# B&R Automation Studio project MotionTestBenchMaster (part 45)

#### HmiInterfacesNew.st
```iecst
ACTION HmiInterfacesNew:
	xAxisInVelocityControl	:= FALSE;

	IF VAR_Machine.iq_stParameter.i_uiAxisSelected >= CST_FillerSubModuleHmiStart AND VAR_Machine.iq_stParameter.i_uiAxisSelected <= CST_FillerSubModuleHmiStart + CST_LastFillerModuleAxis	THEN
		VAR_Machine.stFillerModule.iq_stParameters.i_uiAxisSelected	:= VAR_Machine.iq_stParameter.i_uiAxisSelected - CST_FillerSubModuleHmiStart;
	ELSIF VAR_Machine.iq_stParameter.i_uiAxisSelected >= CST_OutletSubModuleHmiStart AND VAR_Machine.iq_stParameter.i_uiAxisSelected <= CST_OutletSubModuleHmiStart + CST_LastOutletModuleAxis THEN
		VAR_Machine.stOutletModule.iq_stParameters.i_uiAxisSelected	:= VAR_Machine.iq_stParameter.i_uiAxisSelected - CST_OutletSubModuleHmiStart;
	ELSIF VAR_Machine.iq_stParameter.i_uiAxisSelected >= CST_InletSubModuleHmiStart AND VAR_Machine.iq_stParameter.i_uiAxisSelected <= CST_InletSubModuleHmiStart + CST_LastInletModuleAxis THEN
		VAR_Machine.stInletModule.iq_stParameters.i_uiAxisSelected	:= VAR_Machine.iq_stParameter.i_uiAxisSelected - CST_InletSubModuleHmiStart;
	ELSIF VAR_Machine.iq_stParameter.i_uiAxisSelected = CST_MachinePhasingOffset THEN
		VAR_Machine.stMasterModule.iq_stParameters.i_uiAxisSelected	:=	VAR_Machine.iq_stParameter.i_uiAxisSelected;
	END_IF
	////////////////////////////////////////////////

	HMI_MC_GenericAxisDataNew[1].uiDiagCode				:= VAR_Machine.stMasterModule.iq_astSubModuleAxis[CST_MachineMasterAxis].iq_stStatus.q_stMainAxisStatus.q_stInfo.Diag.StatusID.Code;
	HMI_MC_GenericAxisDataNew[1].rLagError				:= FC_DegreeToMm(CFG_MC.Mechanical.MachineStep, VAR_Machine.stMasterModule.iq_astSubModuleAxis[CST_MachineMasterAxis].iq_stStatus.q_stMainAxisStatus.q_rLagError,FALSE);

	HMI_MC_GenericAxisDataNew[1].xMotorWithBrake		:= VAR_Machine.stMasterModule.iq_astSubModuleAxis[CST_MachineMasterAxis].iq_stStatus.q_stMainAxisStatus.q_xMotorWithBrake;
	HMI_MC_GenericAxisDataNew[1].xThirdPartMotor		:= VAR_Machine.stMasterModule.iq_astSubModuleAxis[CST_MachineMasterAxis].iq_stStatus.q_stMainAxisStatus.q_xThirdPartyMotor;
	HMI_MC_GenericAxisDataNew[1].xVelocityControl		:= VAR_Machine.stMasterModule.iq_astSubModuleAxis[CST_MachineMasterAxis].iq_stStatus.q_stMainAxisStatus.q_xVelocityControl;
	HMI_MC_GenericAxisDataNew[1].xInduction				:= VAR_Machine.stMasterModule.iq_astSubModuleAxis[CST_MachineMasterAxis].iq_stStatus.q_stMainAxisStatus.q_xInduction;
	HMI_MC_GenericAxisDataNew[1].rHomingOffset			:= VAR_Machine.stMasterModule.iq_astSubModuleAxis[CST_MachineMasterAxis].iq_stStatus.q_stMainAxisStatus.q_rHomingOffset;

	HMI_MC_GenericAxisDataNew[1].rPosition				:= LREAL_TO_REAL(VAR_Machine.stMasterModule.iq_astSubModuleAxis[CST_MachineMasterAxis].iq_stStatus.q_stMainAxisStatus.q_lrPosition);
	HMI_MC_GenericAxisDataNew[1].rPosition_mm			:= FC_DegreeToMm(CFG_MC.Mechanical.MachineStep,HMI_MC_GenericAxisDataNew[1].rPosition,TRUE);//V1.7.2

	HMI_MC_GenericAxisDataNew[1].rVelocity				:= VAR_Machine.stMasterModule.iq_astSubModuleAxis[CST_MachineMasterAxis].iq_stStatus.q_stMainAxisStatus.q_rVelocity * 10.0;

	HMI_MC_GenericAxisDataNew[1].rTotalPhasingOffset	:= FC_DegreeToMm(CFG_MC.Mechanical.MachineStep,VAR_Machine.stMasterModule.iq_astSubModuleAxis[CST_MachineMasterAxis].iq_stStatus.q_stMainAxisStatus.q_rTotalOffset,FALSE);

	HMI_MC_GenericAxisDataNew[1].xInitialized			:= VAR_Machine.stMasterModule.iq_astSubModuleAxis[CST_MachineMasterAxis].iq_stStatus.q_stMainAxisStatus.q_xInitDone;

	xPhasingRunning									:= VAR_Machine.stMasterModule.iq_astSubModuleAxis[CST_MachineMasterAxis].iq_stStatus.q_stMainAxisStatus.q_xPhasingRunning;

	IF HMI_MC_GenericAxisDataNew[1].xInitialized THEN
		HMI_MC_GenericAxisDataNew[1].xActive				:= VAR_Machine.stMasterModule.iq_astSubModuleAxis[CST_MachineMasterAxis].iq_stStatus.q_stMainAxisStatus.q_xActive;
		HMI_MC_GenericAxisDataNew[1].xBrakeReleased		:= FALSE;
		HMI_MC_GenericAxisDataNew[1].xEnabled;
		HMI_MC_GenericAxisDataNew[1].xFollowingError		:= FALSE;
		HMI_MC_GenericAxisDataNew[1].xHomed				:= FALSE;
		HMI_MC_GenericAxisDataNew[1].xInError				:= VAR_Machine.stMasterModule.iq_astSubModuleAxis[CST_MachineMasterAxis].iq_stStatus.q_stMainAxisStatus.q_xError;
		HMI_MC_GenericAxisDataNew[1].xInPosition			:= VAR_Machine.stMasterModule.iq_astSubModuleAxis[CST_MachineMasterAxis].iq_stStatus.q_stMainAxisStatus.q_xInPosition;
		HMI_MC_GenericAxisDataNew[1].xPowered				:= FALSE;
		HMI_MC_GenericAxisDataNew[1].xReal				:= FALSE;
		HMI_MC_GenericAxisDataNew[1].xRunning				:= FALSE;
		HMI_MC_GenericAxisDataNew[1].xSynchro				:= VAR_Machine.stMasterModule.iq_astSubModuleAxis[CST_MachineMasterAxis].iq_stStatus.q_stMainAxisStatus.q_xSynchronized;
		HMI_MC_GenericAxisDataNew[1].xTorqueError			:= FALSE;
		//			HMI_MC_GenericAxisDataNew[1].xHmiWait				:= FALSE;//V1.7.2
	ELSE
		HMI_MC_GenericAxisDataNew[1].xActive				:= FALSE;
		HMI_MC_GenericAxisDataNew[1].xBrakeReleased		:= FALSE;
		HMI_MC_GenericAxisDataNew[1].xEnabled;
		HMI_MC_GenericAxisDataNew[1].xFollowingError		:= FALSE;
		HMI_MC_GenericAxisDataNew[1].xHomed				:= FALSE;
		HMI_MC_GenericAxisDataNew[1].xInError				:= FALSE;
		HMI_MC_GenericAxisDataNew[1].xInPosition			:= FALSE;
		HMI_MC_GenericAxisDataNew[1].xPowered				:= FALSE;
		HMI_MC_GenericAxisDataNew[1].xReal				:= FALSE;
		HMI_MC_GenericAxisDataNew[1].xRunning				:= FALSE;
		HMI_MC_GenericAxisDataNew[1].xSynchro				:= FALSE;
		HMI_MC_GenericAxisDataNew[1].xTorqueError			:= FALSE;
		//			HMI_MC_GenericAxisDataNew[1].xHmiWait				:= TRUE;//v1.7.2
	END_IF

	FOR HMI_AxisIndex := 2 TO 14 DO //vrma
		//Inlet Axis Motor
		IF HMI_MC_GenericAxisDataNew[HMI_AxisIndex].uiAxisID >= CST_InletSubModuleHmiStart AND HMI_MC_GenericAxisDataNew[HMI_AxisIndex].uiAxisID <= CST_InletSubModuleHmiStart + CST_LastInletModuleAxis THEN

			HMI_MC_GenericAxisDataNew[HMI_AxisIndex].uiDiagCode				:= VAR_Machine.stInletModule.iq_astSubModuleAxis[HMI_MC_GenericAxisDataNew[HMI_AxisIndex].uiAxisID-CST_InletSubModuleHmiStart].iq_stStatus.q_stMainAxisStatus.q_stInfo.Diag.StatusID.Code;
			HMI_MC_GenericAxisDataNew[HMI_AxisIndex].iNextAx_Number;
			HMI_MC_GenericAxisDataNew[HMI_AxisIndex].iPrevAx_Number;
			HMI_MC_GenericAxisDataNew[HMI_AxisIndex].rEncoderTemperature		:= VAR_Machine.stInletModule.iq_astSubModuleAxis[HMI_MC_GenericAxisDataNew[HMI_AxisIndex].uiAxisID-CST_InletSubModuleHmiStart].iq_stStatus.q_stMainAxisStatus.q_rEncoderTemperature;
			HMI_MC_GenericAxisDataNew[HMI_AxisIndex].rMaxTorque;
			HMI_MC_GenericAxisDataNew[HMI_AxisIndex].rLagError				:= FC_DegreeToMm(CFG_MC.Mechanical.MachineStep, VAR_Machine.stInletModule.iq_astSubModuleAxis[HMI_MC_GenericAxisDataNew[HMI_AxisIndex].uiAxisID-CST_InletSubModuleHmiStart].iq_stStatus.q_stMainAxisStatus.q_rLagError, FALSE);

			HMI_MC_GenericAxisDataNew[HMI_AxisIndex].xMotorWithBrake			:= VAR_Machine.stInletModule.iq_astSubModuleAxis[HMI_MC_GenericAxisDataNew[HMI_AxisIndex].uiAxisID-CST_InletSubModuleHmiStart].iq_stStatus.q_stMainAxisStatus.q_xMotorWithBrake;
			HMI_MC_GenericAxisDataNew[HMI_AxisIndex].xThirdPartMotor			:= VAR_Machine.stInletModule.iq_astSubModuleAxis[HMI_MC_GenericAxisDataNew[HMI_AxisIndex].uiAxisID-CST_InletSubModuleHmiStart].iq_stStatus.q_stMainAxisStatus.q_xThirdPartyMotor;
			HMI_MC_GenericAxisDataNew[HMI_AxisIndex].xVelocityControl			:= VAR_Machine.stInletModule.iq_astSubModuleAxis[HMI_MC_GenericAxisDataNew[HMI_AxisIndex].uiAxisID-CST_InletSubModuleHmiStart].iq_stStatus.q_stMainAxisStatus.q_xVelocityControl;
			HMI_MC_GenericAxisDataNew[HMI_AxisIndex].xInduction				:= VAR_Machine.stInletModule.iq_astSubModuleAxis[HMI_MC_GenericAxisDataNew[HMI_AxisIndex].uiAxisID-CST_InletSubModuleHmiStart].iq_stStatus.q_stMainAxisStatus.q_xInduction;
			HMI_MC_GenericAxisDataNew[HMI_AxisIndex].rHomingOffset			:= VAR_Machine.stInletModule.iq_astSubModuleAxis[HMI_MC_GenericAxisDataNew[HMI_AxisIndex].uiAxisID-CST_InletSubModuleHmiStart].iq_stStatus.q_stMainAxisStatus.q_rHomingOffset;

			HMI_MC_GenericAxisDataNew[HMI_AxisIndex].rMotorTemperature		:= VAR_Machine.stInletModule.iq_astSubModuleAxis[HMI_MC_GenericAxisDataNew[HMI_AxisIndex].uiAxisID-CST_InletSubModuleHmiStart].iq_stStatus.q_stMainAxisStatus.q_rMotorTemperature;
			HMI_MC_GenericAxisDataNew[HMI_AxisIndex].rNextAx_Position_mm;
			HMI_MC_GenericAxisDataNew[HMI_AxisIndex].rPosition				:= LREAL_TO_REAL(VAR_Machine.stInletModule.iq_astSubModuleAxis[HMI_MC_GenericAxisDataNew[HMI_AxisIndex].uiAxisID-CST_InletSubModuleHmiStart].iq_stStatus.q_stMainAxisStatus.q_lrPosition);
			HMI_MC_GenericAxisDataNew[HMI_AxisIndex].rPosition_mm			:= FC_DegreeToMm(CFG_MC.Mechanical.MachineStep,HMI_MC_GenericAxisDataNew[HMI_AxisIndex].rPosition,TRUE);//v1.7.2

			HMI_MC_GenericAxisDataNew[HMI_AxisIndex].rPrevAx_Position_mm;
			HMI_MC_GenericAxisDataNew[HMI_AxisIndex].rTorque					:= LREAL_TO_REAL(VAR_Machine.stInletModule.iq_astSubModuleAxis[HMI_MC_GenericAxisDataNew[HMI_AxisIndex].uiAxisID-CST_InletSubModuleHmiStart].iq_stStatus.q_stMainAxisStatus.q_lrTorque);
			HMI_MC_GenericAxisDataNew[HMI_AxisIndex].rVelocity				:= VAR_Machine.stInletModule.iq_astSubModuleAxis[HMI_MC_GenericAxisDataNew[HMI_AxisIndex].uiAxisID-CST_InletSubModuleHmiStart].iq_stStatus.q_stMainAxisStatus.q_rVelocity * 10.0;
			HMI_MC_GenericAxisDataNew[HMI_AxisIndex].rSwitchValue;

			HMI_MC_GenericAxisDataNew[HMI_AxisIndex].rTotalPhasingOffset		:= FC_DegreeToMm(CFG_MC.Mechanical.MachineStep,VAR_Machine.stInletModule.iq_astSubModuleAxis[HMI_MC_GenericAxisDataNew[HMI_AxisIndex].uiAxisID-CST_InletSubModuleHmiStart].iq_stStatus.q_stMainAxisStatus.q_rTotalOffset,FALSE);

			HMI_MC_GenericAxisDataNew[HMI_AxisIndex].xInitialized				:= VAR_Machine.stInletModule.iq_astSubModuleAxis[HMI_MC_GenericAxisDataNew[HMI_AxisIndex].uiAxisID-CST_InletSubModuleHmiStart].iq_stStatus.q_stMainAxisStatus.q_xInitDone;

			xPhasingRunning									:= VAR_Machine.stInletModule.iq_astSubModuleAxis[HMI_MC_GenericAxisDataNew[HMI_AxisIndex].uiAxisID-CST_InletSubModuleHmiStart].iq_stStatus.q_stMainAxisStatus.q_xPhasingRunning;

			IF HMI_MC_GenericAxisDataNew[HMI_AxisIndex].xInitialized THEN
				HMI_MC_GenericAxisDataNew[HMI_AxisIndex].xActive				:= VAR_Machine.stInletModule.iq_astSubModuleAxis[HMI_MC_GenericAxisDataNew[HMI_AxisIndex].uiAxisID-CST_InletSubModuleHmiStart].iq_stStatus.q_stMainAxisStatus.q_xActive;
				HMI_MC_GenericAxisDataNew[HMI_AxisIndex].xBrakeReleased		:= VAR_Machine.stInletModule.iq_astSubModuleAxis[HMI_MC_GenericAxisDataNew[HMI_AxisIndex].uiAxisID-CST_InletSubModuleHmiStart].iq_stStatus.q_stMainAxisStatus.q_xBrakeReleased;
				HMI_MC_GenericAxisDataNew[HMI_AxisIndex].xEnabled;
				HMI_MC_GenericAxisDataNew[HMI_AxisIndex].xFollowingError		:= VAR_Machine.stInletModule.iq_astSubModuleAxis[HMI_MC_GenericAxisDataNew[HMI_AxisIndex].uiAxisID-CST_InletSubModuleHmiStart].iq_stStatus.q_stMainAxisStatus.q_xLagError;
				HMI_MC_GenericAxisDataNew[HMI_AxisIndex].xHomed				:= VAR_Machine.stInletModule.iq_astSubModuleAxis[HMI_MC_GenericAxisDataNew[HMI_AxisIndex].uiAxisID-CST_InletSubModuleHmiStart].iq_stStatus.q_stMainAxisStatus.q_xIsHomed;
				HMI_MC_GenericAxisDataNew[HMI_AxisIndex].xInError				:= VAR_Machine.stInletModule.iq_astSubModuleAxis[HMI_MC_GenericAxisDataNew[HMI_AxisIndex].uiAxisID-CST_InletSubModuleHmiStart].iq_stStatus.q_stMainAxisStatus.q_xError;
				HMI_MC_GenericAxisDataNew[HMI_AxisIndex].xInPosition			:= VAR_Machine.stInletModule.iq_astSubModuleAxis[HMI_MC_GenericAxisDataNew[HMI_AxisIndex].uiAxisID-CST_InletSubModuleHmiStart].iq_stStatus.q_stMainAxisStatus.q_xInPosition;
				HMI_MC_GenericAxisDataNew[HMI_AxisIndex].xPowered				:= VAR_Machine.stInletModule.iq_astSubModuleAxis[HMI_MC_GenericAxisDataNew[HMI_AxisIndex].uiAxisID-CST_InletSubModuleHmiStart].iq_stStatus.q_stMainAxisStatus.q_xPoweredOn;
				HMI_MC_GenericAxisDataNew[HMI_AxisIndex].xReal				:= VAR_Machine.stInletModule.iq_astSubModuleAxis[HMI_MC_GenericAxisDataNew[HMI_AxisIndex].uiAxisID-CST_InletSubModuleHmiStart].iq_stStatus.q_stMainAxisStatus.q_xAxisReal;
				HMI_MC_GenericAxisDataNew[HMI_AxisIndex].xRunning				:= NOT VAR_Machine.stInletModule.iq_astSubModuleAxis[HMI_MC_GenericAxisDataNew[HMI_AxisIndex].uiAxisID-CST_InletSubModuleHmiStart].iq_stStatus.q_stMainAxisStatus.q_xStopped;
				HMI_MC_GenericAxisDataNew[HMI_AxisIndex].xSynchro				:= VAR_Machine.stInletModule.iq_astSubModuleAxis[HMI_MC_GenericAxisDataNew[HMI_AxisIndex].uiAxisID-CST_InletSubModuleHmiStart].iq_stStatus.q_stMainAxisStatus.q_xSynchronized;
				HMI_MC_GenericAxisDataNew[HMI_AxisIndex].xTorqueError			:= VAR_Machine.stInletModule.iq_astSubModuleAxis[HMI_MC_GenericAxisDataNew[HMI_AxisIndex].uiAxisID-CST_InletSubModuleHmiStart].iq_stStatus.q_stMainAxisStatus.q_xTorqueError;
				//HMI_MC_GenericAxisDataNew[HMI_AxisIndex].xHmiWait				:= FALSE;//v1.7.2
			ELSE
				HMI_MC_GenericAxisDataNew[HMI_AxisIndex].xActive				:= FALSE;
				HMI_MC_GenericAxisDataNew[HMI_AxisIndex].xBrakeReleased		:= FALSE;
				HMI_MC_GenericAxisDataNew[HMI_AxisIndex].xEnabled;
				HMI_MC_GenericAxisDataNew[HMI_AxisIndex].xFollowingError		:= FALSE;
				HMI_MC_GenericAxisDataNew[HMI_AxisIndex].xHomed					:= FALSE;
				HMI_MC_GenericAxisDataNew[HMI_AxisIndex].xInError				:= FALSE;
				HMI_MC_GenericAxisDataNew[HMI_AxisIndex].xInPosition			:= FALSE;
				HMI_MC_GenericAxisDataNew[HMI_AxisIndex].xPowered				:= FALSE;
				HMI_MC_GenericAxisDataNew[HMI_AxisIndex].xReal					:= FALSE;
				HMI_MC_GenericAxisDataNew[HMI_AxisIndex].xRunning				:= FALSE;
				HMI_MC_GenericAxisDataNew[HMI_AxisIndex].xSynchro				:= FALSE;
				HMI_MC_GenericAxisDataNew[HMI_AxisIndex].xTorqueError			:= FALSE;
				//				HMI_MC_GenericAxisDataNew[HMI_AxisIndex].xHmiWait				:= TRUE;//v1.7.2
			END_IF
			HMI_MC_GenericAxisData.xBrakeReleased		:= VAR_Machine.stInletModule.iq_astSubModuleAxis[VAR_Machine.stFillerModule.iq_stParameters.i_uiAxisSelected].iq_stStatus.q_stMainAxisStatus.q_xBrakeReleased;//v999 motion test

			HMI_MC_GenericAxisData.xMotorWithBrake	:= VAR_Machine.stInletModule.iq_astSubModuleAxis[VAR_Machine.stFillerModule.iq_stParameters.i_uiAxisSelected].iq_stStatus.q_stMainAxisStatus.q_xMotorWithBrake;//v999 motion test

			xAxisInVelocityControl	:= VAR_Machine.stInletModule.iq_astSubModuleAxis[HMI_MC_GenericAxisDataNew[HMI_AxisIndex].uiAxisID-CST_InletSubModuleHmiStart].iq_stStatus.q_stMainAxisStatus.q_xVelocityControl;
			//Filler Module
		ELSIF HMI_MC_GenericAxisDataNew[HMI_AxisIndex].uiAxisID >= CST_FillerSubModuleHmiStart AND HMI_MC_GenericAxisDataNew[HMI_AxisIndex].uiAxisID <= CST_FillerSubModuleHmiStart + CST_LastFillerModuleAxis THEN
			HMI_MC_GenericAxisDataNew[HMI_AxisIndex].uiDiagCode				:= VAR_Machine.stFillerModule.iq_astSubModuleAxis[HMI_MC_GenericAxisDataNew[HMI_AxisIndex].uiAxisID-CST_FillerSubModuleHmiStart].iq_stStatus.q_stMainAxisStatus.q_stInfo.Diag.StatusID.Code;
			HMI_MC_GenericAxisDataNew[HMI_AxisIndex].iNextAx_Number;
			HMI_MC_GenericAxisDataNew[HMI_AxisIndex].iPrevAx_Number;
			HMI_MC_GenericAxisDataNew[HMI_AxisIndex].rEncoderTemperature		:= VAR_Machine.stFillerModule.iq_astSubModuleAxis[HMI_MC_GenericAxisDataNew[HMI_AxisIndex].uiAxisID-CST_FillerSubModuleHmiStart].iq_stStatus.q_stMainAxisStatus.q_rEncoderTemperature;
			HMI_MC_GenericAxisDataNew[HMI_AxisIndex].rMaxTorque;
			HMI_MC_GenericAxisDataNew[HMI_AxisIndex].rMotorTemperature		:= VAR_Machine.stFillerModule.iq_astSubModuleAxis[HMI_MC_GenericAxisDataNew[HMI_AxisIndex].uiAxisID-CST_FillerSubModuleHmiStart].iq_stStatus.q_stMainAxisStatus.q_rMotorTemperature;
			HMI_MC_GenericAxisDataNew[HMI_AxisIndex].rNextAx_Position_mm;
			HMI_MC_GenericAxisDataNew[HMI_AxisIndex].rPosition				:= LREAL_TO_REAL(VAR_Machine.stFillerModule.iq_astSubModuleAxis[HMI_MC_GenericAxisDataNew[HMI_AxisIndex].uiAxisID-CST_FillerSubModuleHmiStart].iq_stStatus.q_stMainAxisStatus.q_lrPosition);
			HMI_MC_GenericAxisDataNew[HMI_AxisIndex].rPosition_mm			:= FC_DegreeToMm(CFG_MC.Mechanical.MachineStep,HMI_MC_GenericAxisDataNew[HMI_AxisIndex].rPosition,TRUE);//v1.7.2

			HMI_MC_GenericAxisDataNew[HMI_AxisIndex].xMotorWithBrake			:= VAR_Machine.stFillerModule.iq_astSubModuleAxis[HMI_MC_GenericAxisDataNew[HMI_AxisIndex].uiAxisID-CST_FillerSubModuleHmiStart].iq_stStatus.q_stMainAxisStatus.q_xMotorWithBrake;
			HMI_MC_GenericAxisDataNew[HMI_AxisIndex].xThirdPartMotor			:= VAR_Machine.stFillerModule.iq_astSubModuleAxis[HMI_MC_GenericAxisDataNew[HMI_AxisIndex].uiAxisID-CST_FillerSubModuleHmiStart].iq_stStatus.q_stMainAxisStatus.q_xThirdPartyMotor;
			HMI_MC_GenericAxisDataNew[HMI_AxisIndex].xVelocityControl			:= VAR_Machine.stFillerModule.iq_astSubModuleAxis[HMI_MC_GenericAxisDataNew[HMI_AxisIndex].uiAxisID-CST_FillerSubModuleHmiStart].iq_stStatus.q_stMainAxisStatus.q_xVelocityControl;
			HMI_MC_GenericAxisDataNew[HMI_AxisIndex].xInduction				:= VAR_Machine.stFillerModule.iq_astSubModuleAxis[HMI_MC_GenericAxisDataNew[HMI_AxisIndex].uiAxisID-CST_FillerSubModuleHmiStart].iq_stStatus.q_stMainAxisStatus.q_xInduction;
			HMI_MC_GenericAxisDataNew[HMI_AxisIndex].rHomingOffset			:= VAR_Machine.stFillerModule.iq_astSubModuleAxis[HMI_MC_GenericAxisDataNew[HMI_AxisIndex].uiAxisID-CST_FillerSubModuleHmiStart].iq_stStatus.q_stMainAxisStatus.q_rHomingOffset;

			HMI_MC_GenericAxisDataNew[HMI_AxisIndex].rTotalPhasingOffset		:= FC_DegreeToMm(CFG_MC.Mechanical.MachineStep,VAR_Machine.stFillerModule.iq_astSubModuleAxis[HMI_MC_GenericAxisDataNew[HMI_AxisIndex].uiAxisID-CST_FillerSubModuleHmiStart].iq_stStatus.q_stMainAxisStatus.q_rTotalOffset, FALSE);

			HMI_MC_GenericAxisDataNew[HMI_AxisIndex].rLagError				:= FC_DegreeToMm(CFG_MC.Mechanical.MachineStep, VAR_Machine.stFillerModule.iq_astSubModuleAxis[HMI_MC_GenericAxisDataNew[HMI_AxisIndex].uiAxisID-CST_FillerSubModuleHmiStart].iq_stStatus.q_stMainAxisStatus.q_rLagError, FALSE);

			HMI_MC_GenericAxisDataNew[HMI_AxisIndex].rPrevAx_Position_mm;
			HMI_MC_GenericAxisDataNew[HMI_AxisIndex].rTorque					:= LREAL_TO_REAL(VAR_Machine.stFillerModule.iq_astSubModuleAxis[HMI_MC_GenericAxisDataNew[HMI_AxisIndex].uiAxisID-CST_FillerSubModuleHmiStart].iq_stStatus.q_stMainAxisStatus.q_lrTorque);
			HMI_MC_GenericAxisDataNew[HMI_AxisIndex].rVelocity				:= VAR_Machine.stFillerModule.iq_astSubModuleAxis[HMI_MC_GenericAxisDataNew[HMI_AxisIndex].uiAxisID-CST_FillerSubModuleHmiStart].iq_stStatus.q_stMainAxisStatus.q_rVelocity * 10.0;
			HMI_MC_GenericAxisDataNew[HMI_AxisIndex].rSwitchValue;

			HMI_MC_GenericAxisDataNew[HMI_AxisIndex].xInitialized				:= VAR_Machine.stFillerModule.iq_astSubModuleAxis[HMI_MC_GenericAxisDataNew[HMI_AxisIndex].uiAxisID-CST_FillerSubModuleHmiStart].iq_stStatus.q_stMainAxisStatus.q_xInitDone;

			xPhasingRunning									:= VAR_Machine.stFillerModule.iq_astSubModuleAxis[HMI_MC_GenericAxisDataNew[HMI_AxisIndex].uiAxisID-CST_FillerSubModuleHmiStart].iq_stStatus.q_stMainAxisStatus.q_xPhasingRunning;

			IF HMI_MC_GenericAxisDataNew[HMI_AxisIndex].xInitialized THEN
				HMI_MC_GenericAxisDataNew[HMI_AxisIndex].xActive				:= VAR_Machine.stFillerModule.iq_astSubModuleAxis[HMI_MC_GenericAxisDataNew[HMI_AxisIndex].uiAxisID-CST_FillerSubModuleHmiStart].iq_stStatus.q_stMainAxisStatus.q_xActive;
				HMI_MC_GenericAxisDataNew[HMI_AxisIndex].xBrakeReleased		:= VAR_Machine.stFillerModule.iq_astSubModuleAxis[HMI_MC_GenericAxisDataNew[HMI_AxisIndex].uiAxisID-CST_FillerSubModuleHmiStart].iq_stStatus.q_stMainAxisStatus.q_xBrakeReleased;
				HMI_MC_GenericAxisDataNew[HMI_AxisIndex].xEnabled;
				HMI_MC_GenericAxisDataNew[HMI_AxisIndex].xFollowingError		:= VAR_Machine.stFillerModule.iq_astSubModuleAxis[HMI_MC_GenericAxisDataNew[HMI_AxisIndex].uiAxisID-CST_FillerSubModuleHmiStart].iq_stStatus.q_stMainAxisStatus.q_xLagError;
				HMI_MC_GenericAxisDataNew[HMI_AxisIndex].xHomed				:= VAR_Machine.stFillerModule.iq_astSubModuleAxis[HMI_MC_GenericAxisDataNew[HMI_AxisIndex].uiAxisID-CST_FillerSubModuleHmiStart].iq_stStatus.q_stMainAxisStatus.q_xIsHomed;
				HMI_MC_GenericAxisDataNew[HMI_AxisIndex].xInError				:= VAR_Machine.stFillerModule.iq_astSubModuleAxis[HMI_MC_GenericAxisDataNew[HMI_AxisIndex].uiAxisID-CST_FillerSubModuleHmiStart].iq_stStatus.q_stMainAxisStatus.q_xError;
				HMI_MC_GenericAxisDataNew[HMI_AxisIndex].xInPosition			:= VAR_Machine.stFillerModule.iq_astSubModuleAxis[HMI_MC_GenericAxisDataNew[HMI_AxisIndex].uiAxisID-CST_FillerSubModuleHmiStart].iq_stStatus.q_stMainAxisStatus.q_xInPosition;
				HMI_MC_GenericAxisDataNew[HMI_AxisIndex].xPowered				:= VAR_Machine.stFillerModule.iq_astSubModuleAxis[HMI_MC_GenericAxisDataNew[HMI_AxisIndex].uiAxisID-CST_FillerSubModuleHmiStart].iq_stStatus.q_stMainAxisStatus.q_xPoweredOn;
				HMI_MC_GenericAxisDataNew[HMI_AxisIndex].xReal				:= VAR_Machine.stFillerModule.iq_astSubModuleAxis[HMI_MC_GenericAxisDataNew[HMI_AxisIndex].uiAxisID-CST_FillerSubModuleHmiStart].iq_stStatus.q_stMainAxisStatus.q_xAxisReal;
				HMI_MC_GenericAxisDataNew[HMI_AxisIndex].xRunning				:= NOT VAR_Machine.stFillerModule.iq_astSubModuleAxis[HMI_MC_GenericAxisDataNew[HMI_AxisIndex].uiAxisID-CST_FillerSubModuleHmiStart].iq_stStatus.q_stMainAxisStatus.q_xStopped;
				HMI_MC_GenericAxisDataNew[HMI_AxisIndex].xSynchro				:= VAR_Machine.stFillerModule.iq_astSubModuleAxis[HMI_MC_GenericAxisDataNew[HMI_AxisIndex].uiAxisID-CST_FillerSubModuleHmiStart].iq_stStatus.q_stMainAxisStatus.q_xSynchronized;
				HMI_MC_GenericAxisDataNew[HMI_AxisIndex].xTorqueError			:= VAR_Machine.stFillerModule.iq_astSubModuleAxis[HMI_MC_GenericAxisDataNew[HMI_AxisIndex].uiAxisID-CST_FillerSubModuleHmiStart].iq_stStatus.q_stMainAxisStatus.q_xTorqueError;
				//HMI_MC_GenericAxisDataNew[HMI_AxisIndex].xHmiWait				:= FALSE;//v1.7.2
			ELSE
				HMI_MC_GenericAxisDataNew[HMI_AxisIndex].xActive				:= FALSE;
				HMI_MC_GenericAxisDataNew[HMI_AxisIndex].xBrakeReleased		:= FALSE;
				HMI_MC_GenericAxisDataNew[HMI_AxisIndex].xEnabled;
				HMI_MC_GenericAxisDataNew[HMI_AxisIndex].xFollowingError		:= FALSE;
				HMI_MC_GenericAxisDataNew[HMI_AxisIndex].xHomed				:= FALSE;
				HMI_MC_GenericAxisDataNew[HMI_AxisIndex].xInError				:= FALSE;
				HMI_MC_GenericAxisDataNew[HMI_AxisIndex].xInPosition			:= FALSE;
				HMI_MC_GenericAxisDataNew[HMI_AxisIndex].xPowered				:= FALSE;
				HMI_MC_GenericAxisDataNew[HMI_AxisIndex].xReal				:= FALSE;
				HMI_MC_GenericAxisDataNew[HMI_AxisIndex].xRunning				:= FALSE;
				HMI_MC_GenericAxisDataNew[HMI_AxisIndex].xSynchro				:= FALSE;
				HMI_MC_GenericAxisDataNew[HMI_AxisIndex].xTorqueError			:= FALSE;
				//HMI_MC_GenericAxisDataNew[HMI_AxisIndex].xHmiWait				:= TRUE;//v1.7.2
			END_IF
			HMI_MC_GenericAxisData.xBrakeReleased		:= VAR_Machine.stFillerModule.iq_astSubModuleAxis[VAR_Machine.stFillerModule.iq_stParameters.i_uiAxisSelected].iq_stStatus.q_stMainAxisStatus.q_xBrakeReleased;//v999 motion test

			HMI_MC_GenericAxisData.xMotorWithBrake	:= VAR_Machine.stFillerModule.iq_astSubModuleAxis[VAR_Machine.stFillerModule.iq_stParameters.i_uiAxisSelected].iq_stStatus.q_stMainAxisStatus.q_xMotorWithBrake;//v999 motion test

			xAxisInVelocityControl	:= VAR_Machine.stFillerModule.iq_astSubModuleAxis[HMI_MC_GenericAxisDataNew[HMI_AxisIndex].uiAxisID-CST_FillerSubModuleHmiStart].iq_stStatus.q_stMainAxisStatus.q_xVelocityControl;
			//Outlet Module
		ELSIF HMI_MC_GenericAxisDataNew[HMI_AxisIndex].uiAxisID >= CST_OutletSubModuleHmiStart AND HMI_MC_GenericAxisDataNew[HMI_AxisIndex].uiAxisID <= CST_OutletSubModuleHmiStart + CST_LastOutletModuleAxis THEN
			HMI_MC_GenericAxisDataNew[HMI_AxisIndex].uiDiagCode					:= VAR_Machine.stOutletModule.iq_astSubModuleAxis[HMI_MC_GenericAxisDataNew[HMI_AxisIndex].uiAxisID - CST_OutletSubModuleHmiStart].iq_stStatus.q_stMainAxisStatus.q_stInfo.Diag.StatusID.Code;
			HMI_MC_GenericAxisDataNew[HMI_AxisIndex].iNextAx_Number;
			HMI_MC_GenericAxisDataNew[HMI_AxisIndex].iPrevAx_Number;
			HMI_MC_GenericAxisDataNew[HMI_AxisIndex].rEncoderTemperature		:= VAR_Machine.stOutletModule.iq_astSubModuleAxis[HMI_MC_GenericAxisDataNew[HMI_AxisIndex].uiAxisID - CST_OutletSubModuleHmiStart].iq_stStatus.q_stMainAxisStatus.q_rEncoderTemperature;
			HMI_MC_GenericAxisDataNew[HMI_AxisIndex].rMaxTorque;
			HMI_MC_GenericAxisDataNew[HMI_AxisIndex].rLagError					:= FC_DegreeToMm(CFG_MC.Mechanical.MachineStep, VAR_Machine.stOutletModule.iq_astSubModuleAxis[HMI_MC_GenericAxisDataNew[HMI_AxisIndex].uiAxisID - CST_OutletSubModuleHmiStart].iq_stStatus.q_stMainAxisStatus.q_rLagError, FALSE);

			HMI_MC_GenericAxisDataNew[HMI_AxisIndex].xMotorWithBrake			:= VAR_Machine.stOutletModule.iq_astSubModuleAxis[HMI_MC_GenericAxisDataNew[HMI_AxisIndex].uiAxisID - CST_OutletSubModuleHmiStart].iq_stStatus.q_stMainAxisStatus.q_xMotorWithBrake;
			HMI_MC_GenericAxisDataNew[HMI_AxisIndex].xThirdPartMotor			:= VAR_Machine.stOutletModule.iq_astSubModuleAxis[HMI_MC_GenericAxisDataNew[HMI_AxisIndex].uiAxisID - CST_OutletSubModuleHmiStart].iq_stStatus.q_stMainAxisStatus.q_xThirdPartyMotor;
			HMI_MC_GenericAxisDataNew[HMI_AxisIndex].xVelocityControl			:= VAR_Machine.stOutletModule.iq_astSubModuleAxis[HMI_MC_GenericAxisDataNew[HMI_AxisIndex].uiAxisID - CST_OutletSubModuleHmiStart].iq_stStatus.q_stMainAxisStatus.q_xVelocityControl;
			HMI_MC_GenericAxisDataNew[HMI_AxisIndex].xInduction					:= VAR_Machine.stOutletModule.iq_astSubModuleAxis[HMI_MC_GenericAxisDataNew[HMI_AxisIndex].uiAxisID - CST_OutletSubModuleHmiStart].iq_stStatus.q_stMainAxisStatus.q_xInduction;
			HMI_MC_GenericAxisDataNew[HMI_AxisIndex].rHomingOffset				:= VAR_Machine.stOutletModule.iq_astSubModuleAxis[HMI_MC_GenericAxisDataNew[HMI_AxisIndex].uiAxisID - CST_OutletSubModuleHmiStart].iq_stStatus.q_stMainAxisStatus.q_rHomingOffset;

			HMI_MC_GenericAxisDataNew[HMI_AxisIndex].rMotorTemperature			:= VAR_Machine.stOutletModule.iq_astSubModuleAxis[HMI_MC_GenericAxisDataNew[HMI_AxisIndex].uiAxisID - CST_OutletSubModuleHmiStart].iq_stStatus.q_stMainAxisStatus.q_rMotorTemperature;
			HMI_MC_GenericAxisDataNew[HMI_AxisIndex].rNextAx_Position_mm;
			HMI_MC_GenericAxisDataNew[HMI_AxisIndex].rPosition					:= LREAL_TO_REAL(VAR_Machine.stOutletModule.iq_astSubModuleAxis[HMI_MC_GenericAxisDataNew[HMI_AxisIndex].uiAxisID - CST_OutletSubModuleHmiStart].iq_stStatus.q_stMainAxisStatus.q_lrPosition);
			HMI_MC_GenericAxisDataNew[HMI_AxisIndex].rPosition_mm				:= FC_DegreeToMm(CFG_MC.Mechanical.MachineStep,HMI_MC_GenericAxisDataNew[HMI_AxisIndex].rPosition,TRUE);//v1.7.2

			HMI_MC_GenericAxisDataNew[HMI_AxisIndex].rPrevAx_Position_mm;
			HMI_MC_GenericAxisDataNew[HMI_AxisIndex].rTorque					:= LREAL_TO_REAL(VAR_Machine.stOutletModule.iq_astSubModuleAxis[HMI_MC_GenericAxisDataNew[HMI_AxisIndex].uiAxisID - CST_OutletSubModuleHmiStart].iq_stStatus.q_stMainAxisStatus.q_lrTorque);
			HMI_MC_GenericAxisDataNew[HMI_AxisIndex].rVelocity					:= VAR_Machine.stOutletModule.iq_astSubModuleAxis[HMI_MC_GenericAxisDataNew[HMI_AxisIndex].uiAxisID - CST_OutletSubModuleHmiStart].iq_stStatus.q_stMainAxisStatus.q_rVelocity * 10.0;
			HMI_MC_GenericAxisDataNew[HMI_AxisIndex].rSwitchValue;

			HMI_MC_GenericAxisDataNew[HMI_AxisIndex].rTotalPhasingOffset		:= FC_DegreeToMm(CFG_MC.Mechanical.MachineStep,VAR_Machine.stOutletModule.iq_astSubModuleAxis[HMI_MC_GenericAxisDataNew[HMI_AxisIndex].uiAxisID - CST_OutletSubModuleHmiStart].iq_stStatus.q_stMainAxisStatus.q_rTotalOffset,FALSE);

			HMI_MC_GenericAxisDataNew[HMI_AxisIndex].xInitialized				:= VAR_Machine.stOutletModule.iq_astSubModuleAxis[HMI_MC_GenericAxisDataNew[HMI_AxisIndex].uiAxisID - CST_OutletSubModuleHmiStart].iq_stStatus.q_stMainAxisStatus.q_xInitDone;

			xPhasingRunning														:= VAR_Machine.stOutletModule.iq_astSubModuleAxis[HMI_MC_GenericAxisDataNew[HMI_AxisIndex].uiAxisID - CST_OutletSubModuleHmiStart].iq_stStatus.q_stMainAxisStatus.q_xPhasingRunning;

			IF HMI_MC_GenericAxisDataNew[HMI_AxisIndex].xInitialized THEN
				HMI_MC_GenericAxisDataNew[HMI_AxisIndex].xActive				:= VAR_Machine.stOutletModule.iq_astSubModuleAxis[HMI_MC_GenericAxisDataNew[HMI_AxisIndex].uiAxisID - CST_OutletSubModuleHmiStart].iq_stStatus.q_stMainAxisStatus.q_xActive;
				HMI_MC_GenericAxisDataNew[HMI_AxisIndex].xBrakeReleased			:= VAR_Machine.stOutletModule.iq_astSubModuleAxis[HMI_MC_GenericAxisDataNew[HMI_AxisIndex].uiAxisID - CST_OutletSubModuleHmiStart].iq_stStatus.q_stMainAxisStatus.q_xBrakeReleased;
				HMI_MC_GenericAxisDataNew[HMI_AxisIndex].xEnabled;
				HMI_MC_GenericAxisDataNew[HMI_AxisIndex].xFollowingError		:= VAR_Machine.stOutletModule.iq_astSubModuleAxis[HMI_MC_GenericAxisDataNew[HMI_AxisIndex].uiAxisID - CST_OutletSubModuleHmiStart].iq_stStatus.q_stMainAxisStatus.q_xLagError;
				HMI_MC_GenericAxisDataNew[HMI_AxisIndex].xHomed					:= VAR_Machine.stOutletModule.iq_astSubModuleAxis[HMI_MC_GenericAxisDataNew[HMI_AxisIndex].uiAxisID - CST_OutletSubModuleHmiStart].iq_stStatus.q_stMainAxisStatus.q_xIsHomed;
				HMI_MC_GenericAxisDataNew[HMI_AxisIndex].xInError				:= VAR_Machine.stOutletModule.iq_astSubModuleAxis[HMI_MC_GenericAxisDataNew[HMI_AxisIndex].uiAxisID - CST_OutletSubModuleHmiStart].iq_stStatus.q_stMainAxisStatus.q_xError;
				HMI_MC_GenericAxisDataNew[HMI_AxisIndex].xInPosition			:= VAR_Machine.stOutletModule.iq_astSubModuleAxis[HMI_MC_GenericAxisDataNew[HMI_AxisIndex].uiAxisID - CST_OutletSubModuleHmiStart].iq_stStatus.q_stMainAxisStatus.q_xInPosition;
				HMI_MC_GenericAxisDataNew[HMI_AxisIndex].xPowered				:= VAR_Machine.stOutletModule.iq_astSubModuleAxis[HMI_MC_GenericAxisDataNew[HMI_AxisIndex].uiAxisID - CST_OutletSubModuleHmiStart].iq_stStatus.q_stMainAxisStatus.q_xPoweredOn;
				HMI_MC_GenericAxisDataNew[HMI_AxisIndex].xReal					:= VAR_Machine.stOutletModule.iq_astSubModuleAxis[HMI_MC_GenericAxisDataNew[HMI_AxisIndex].uiAxisID - CST_OutletSubModuleHmiStart].iq_stStatus.q_stMainAxisStatus.q_xAxisReal;
				HMI_MC_GenericAxisDataNew[HMI_AxisIndex].xRunning				:= NOT VAR_Machine.stOutletModule.iq_astSubModuleAxis[HMI_MC_GenericAxisDataNew[HMI_AxisIndex].uiAxisID - CST_OutletSubModuleHmiStart].iq_stStatus.q_stMainAxisStatus.q_xStopped;
				HMI_MC_GenericAxisDataNew[HMI_AxisIndex].xSynchro				:= VAR_Machine.stOutletModule.iq_astSubModuleAxis[HMI_MC_GenericAxisDataNew[HMI_AxisIndex].uiAxisID - CST_OutletSubModuleHmiStart].iq_stStatus.q_stMainAxisStatus.q_xSynchronized;
				HMI_MC_GenericAxisDataNew[HMI_AxisIndex].xTorqueError			:= VAR_Machine.stOutletModule.iq_astSubModuleAxis[HMI_MC_GenericAxisDataNew[HMI_AxisIndex].uiAxisID - CST_OutletSubModuleHmiStart].iq_stStatus.q_stMainAxisStatus.q_xTorqueError;
				//HMI_MC_GenericAxisDataNew[HMI_AxisIndex].xHmiWait				:= FALSE;
			ELSE
				HMI_MC_GenericAxisDataNew[HMI_AxisIndex].xActive				:= FALSE;
				HMI_MC_GenericAxisDataNew[HMI_AxisIndex].xBrakeReleased			:= FALSE;
				HMI_MC_GenericAxisDataNew[HMI_AxisIndex].xEnabled;
				HMI_MC_GenericAxisDataNew[HMI_AxisIndex].xFollowingError		:= FALSE;
				HMI_MC_GenericAxisDataNew[HMI_AxisIndex].xHomed					:= FALSE;
				HMI_MC_GenericAxisDataNew[HMI_AxisIndex].xInError				:= FALSE;
				HMI_MC_GenericAxisDataNew[HMI_AxisIndex].xInPosition			:= FALSE;
				HMI_MC_GenericAxisDataNew[HMI_AxisIndex].xPowered				:= FALSE;
				HMI_MC_GenericAxisDataNew[HMI_AxisIndex].xReal					:= FALSE;
				HMI_MC_GenericAxisDataNew[HMI_AxisIndex].xRunning				:= FALSE;
				HMI_MC_GenericAxisDataNew[HMI_AxisIndex].xSynchro				:= FALSE;
				HMI_MC_GenericAxisDataNew[HMI_AxisIndex].xTorqueError			:= FALSE;
				//HMI_MC_GenericAxisDataNew[HMI_AxisIndex].xHmiWait				:= TRUE;
			END_IF
			HMI_MC_GenericAxisData.xBrakeReleased		:= VAR_Machine.stOutletModule.iq_astSubModuleAxis[VAR_Machine.stOutletModule.iq_stParameters.i_uiAxisSelected].iq_stStatus.q_stMainAxisStatus.q_xBrakeReleased;//v999 motion test

			HMI_MC_GenericAxisData.xMotorWithBrake	:=  VAR_Machine.stOutletModule.iq_astSubModuleAxis[VAR_Machine.stOutletModule.iq_stParameters.i_uiAxisSelected].iq_stStatus.q_stMainAxisStatus.q_xBrakeReleased;//v999 motion test
			;

			xAxisInVelocityControl	:= VAR_Machine.stOutletModule.iq_astSubModuleAxis[HMI_MC_GenericAxisDataNew[HMI_AxisIndex].uiAxisID - CST_OutletSubModuleHmiStart].iq_stStatus.q_stMainAxisStatus.q_xVelocityControl;

		END_IF
	END_FOR

	IF VAR_Machine.stFillerModule.iq_stStatus.q_xInitDone AND  VAR_Machine.stInletModule.iq_stStatus.q_xInitDone AND VAR_Machine.stOutletModule.iq_stStatus.q_xInitDone THEN//v1.7.2
		HMI_MC_GenericAxisData.xHmiWait										:= FALSE ;//v1.7.2
	ELSE //v1.7.2
		HMI_MC_GenericAxisData.xHmiWait										:= TRUE;//v1.7.2
		END_IF//v1.7.2

	/////////////////////////////////////////////////
	HMI_MC_EncoderDiagnostic.Present 									:= CFG_MC.Generic.SyncroPar.ExternalEncoder;
	HMI_MC_EncoderDiagnostic.ModuleOK 									:= MC_InputOutput.Network.Machine.Commands.MasterEncoderPositionValid;
	HMI_MC_EncoderDiagnostic.Value 										:= ITC_Motion_ExtEnc;

	HMI_MC_GenericAxisData.rPosition									:= LREAL_TO_REAL(VAR_Machine.stFillerModule.iq_astSubModuleAxis[15].iq_stStatus.q_stMainAxisStatus.q_lrPosition);//V4.A.A.1.7.0
	END_ACTION
```

#### HmiInterfaces.st
```iecst
ACTION HmiInterfaces:
	xAxisInVelocityControl	:= FALSE;

	IF VAR_Machine.iq_stParameter.i_uiAxisSelected >= CST_FillerSubModuleHmiStart AND VAR_Machine.iq_stParameter.i_uiAxisSelected <= CST_FillerSubModuleHmiStart + CST_LastFillerModuleAxis	THEN

		VAR_Machine.stFillerModule.iq_stParameters.i_uiAxisSelected	:= VAR_Machine.iq_stParameter.i_uiAxisSelected - CST_FillerSubModuleHmiStart;

		HMI_MC_GenericAxisData.uiDiagCode				:= VAR_Machine.stFillerModule.iq_astSubModuleAxis[VAR_Machine.stFillerModule.iq_stParameters.i_uiAxisSelected].iq_stStatus.q_stMainAxisStatus.q_stInfo.Diag.StatusID.Code;
		HMI_MC_GenericAxisData.iNextAx_Number;
		HMI_MC_GenericAxisData.iPrevAx_Number;
		HMI_MC_GenericAxisData.rEncoderTemperature		:= VAR_Machine.stFillerModule.iq_astSubModuleAxis[VAR_Machine.stFillerModule.iq_stParameters.i_uiAxisSelected].iq_stStatus.q_stMainAxisStatus.q_rEncoderTemperature;
		HMI_MC_GenericAxisData.rMaxTorque;
		HMI_MC_GenericAxisData.rMotorTemperature		:= VAR_Machine.stFillerModule.iq_astSubModuleAxis[VAR_Machine.stFillerModule.iq_stParameters.i_uiAxisSelected].iq_stStatus.q_stMainAxisStatus.q_rMotorTemperature;
		HMI_MC_GenericAxisData.rNextAx_Position_mm;
		HMI_MC_GenericAxisData.rPosition				:= LREAL_TO_REAL(VAR_Machine.stFillerModule.iq_astSubModuleAxis[VAR_Machine.stFillerModule.iq_stParameters.i_uiAxisSelected].iq_stStatus.q_stMainAxisStatus.q_lrPosition);
		HMI_MC_GenericAxisData.rPosition_mm				:= FC_DegreeToMm(CFG_MC.Mechanical.MachineStep, HMI_MC_GenericAxisData.rPosition, TRUE);

		HMI_MC_GenericAxisData.xMotorWithBrake			:= VAR_Machine.stFillerModule.iq_astSubModuleAxis[VAR_Machine.stFillerModule.iq_stParameters.i_uiAxisSelected].iq_stStatus.q_stMainAxisStatus.q_xMotorWithBrake;
		HMI_MC_GenericAxisData.xThirdPartMotor			:= VAR_Machine.stFillerModule.iq_astSubModuleAxis[VAR_Machine.stFillerModule.iq_stParameters.i_uiAxisSelected].iq_stStatus.q_stMainAxisStatus.q_xThirdPartyMotor;
		HMI_MC_GenericAxisData.xVelocityControl			:= VAR_Machine.stFillerModule.iq_astSubModuleAxis[VAR_Machine.stFillerModule.iq_stParameters.i_uiAxisSelected].iq_stStatus.q_stMainAxisStatus.q_xVelocityControl;
		HMI_MC_GenericAxisData.xInduction				:= VAR_Machine.stFillerModule.iq_astSubModuleAxis[VAR_Machine.stFillerModule.iq_stParameters.i_uiAxisSelected].iq_stStatus.q_stMainAxisStatus.q_xInduction;
		HMI_MC_GenericAxisData.rHomingOffset			:= VAR_Machine.stFillerModule.iq_astSubModuleAxis[VAR_Machine.stFillerModule.iq_stParameters.i_uiAxisSelected].iq_stStatus.q_stMainAxisStatus.q_rHomingOffset;

		HMI_MC_GenericAxisData.rTotalPhasingOffset		:= FC_DegreeToMm(CFG_MC.Mechanical.MachineStep,VAR_Machine.stFillerModule.iq_astSubModuleAxis[VAR_Machine.stFillerModule.iq_stParameters.i_uiAxisSelected].iq_stStatus.q_stMainAxisStatus.q_rTotalOffset, FALSE);

		HMI_MC_GenericAxisData.rLagError				:= FC_DegreeToMm(CFG_MC.Mechanical.MachineStep, VAR_Machine.stFillerModule.iq_astSubModuleAxis[VAR_Machine.stFillerModule.iq_stParameters.i_uiAxisSelected].iq_stStatus.q_stMainAxisStatus.q_rLagError, FALSE);

		HMI_MC_GenericAxisData.rPrevAx_Position_mm;
		HMI_MC_GenericAxisData.rTorque					:= LREAL_TO_REAL(VAR_Machine.stFillerModule.iq_astSubModuleAxis[VAR_Machine.stFillerModule.iq_stParameters.i_uiAxisSelected].iq_stStatus.q_stMainAxisStatus.q_lrTorque);
		HMI_MC_GenericAxisData.rVelocity				:= VAR_Machine.stFillerModule.iq_astSubModuleAxis[VAR_Machine.stFillerModule.iq_stParameters.i_uiAxisSelected].iq_stStatus.q_stMainAxisStatus.q_rVelocity * 10.0;
		HMI_MC_GenericAxisData.rSwitchValue;

		HMI_MC_GenericAxisData.xInitialized				:= VAR_Machine.stFillerModule.iq_astSubModuleAxis[VAR_Machine.stFillerModule.iq_stParameters.i_uiAxisSelected].iq_stStatus.q_stMainAxisStatus.q_xInitDone;

		xPhasingRunning									:= VAR_Machine.stFillerModule.iq_astSubModuleAxis[VAR_Machine.stFillerModule.iq_stParameters.i_uiAxisSelected].iq_stStatus.q_stMainAxisStatus.q_xPhasingRunning;

		IF HMI_MC_GenericAxisData.xInitialized THEN
			HMI_MC_GenericAxisData.xActive				:= VAR_Machine.stFillerModule.iq_astSubModuleAxis[VAR_Machine.stFillerModule.iq_stParameters.i_uiAxisSelected].iq_stStatus.q_stMainAxisStatus.q_xActive;
			HMI_MC_GenericAxisData.xBrakeReleased		:= VAR_Machine.stFillerModule.iq_astSubModuleAxis[VAR_Machine.stFillerModule.iq_stParameters.i_uiAxisSelected].iq_stStatus.q_stMainAxisStatus.q_xBrakeReleased;
			HMI_MC_GenericAxisData.xEnabled;
			HMI_MC_GenericAxisData.xFollowingError		:= VAR_Machine.stFillerModule.iq_astSubModuleAxis[VAR_Machine.stFillerModule.iq_stParameters.i_uiAxisSelected].iq_stStatus.q_stMainAxisStatus.q_xLagError;
			HMI_MC_GenericAxisData.xHomed				:= VAR_Machine.stFillerModule.iq_astSubModuleAxis[VAR_Machine.stFillerModule.iq_stParameters.i_uiAxisSelected].iq_stStatus.q_stMainAxisStatus.q_xIsHomed;
			HMI_MC_GenericAxisData.xInError				:= VAR_Machine.stFillerModule.iq_astSubModuleAxis[VAR_Machine.stFillerModule.iq_stParameters.i_uiAxisSelected].iq_stStatus.q_stMainAxisStatus.q_xError;
			HMI_MC_GenericAxisData.xInPosition			:= VAR_Machine.stFillerModule.iq_astSubModuleAxis[VAR_Machine.stFillerModule.iq_stParameters.i_uiAxisSelected].iq_stStatus.q_stMainAxisStatus.q_xInPosition;
			HMI_MC_GenericAxisData.xPowered				:= VAR_Machine.stFillerModule.iq_astSubModuleAxis[VAR_Machine.stFillerModule.iq_stParameters.i_uiAxisSelected].iq_stStatus.q_stMainAxisStatus.q_xPoweredOn;
			HMI_MC_GenericAxisData.xReal				:= VAR_Machine.stFillerModule.iq_astSubModuleAxis[VAR_Machine.stFillerModule.iq_stParameters.i_uiAxisSelected].iq_stStatus.q_stMainAxisStatus.q_xAxisReal;
			HMI_MC_GenericAxisData.xRunning				:= NOT VAR_Machine.stFillerModule.iq_astSubModuleAxis[VAR_Machine.stFillerModule.iq_stParameters.i_uiAxisSelected].iq_stStatus.q_stMainAxisStatus.q_xStopped;
			HMI_MC_GenericAxisData.xSynchro				:= VAR_Machine.stFillerModule.iq_astSubModuleAxis[VAR_Machine.stFillerModule.iq_stParameters.i_uiAxisSelected].iq_stStatus.q_stMainAxisStatus.q_xSynchronized;
			HMI_MC_GenericAxisData.xTorqueError			:= VAR_Machine.stFillerModule.iq_astSubModuleAxis[VAR_Machine.stFillerModule.iq_stParameters.i_uiAxisSelected].iq_stStatus.q_stMainAxisStatus.q_xTorqueError;
			HMI_MC_GenericAxisData.xHmiWait				:= FALSE;
		ELSE
			HMI_MC_GenericAxisData.xActive				:= FALSE;
			HMI_MC_GenericAxisData.xBrakeReleased		:= FALSE;
			HMI_MC_GenericAxisData.xEnabled;
			HMI_MC_GenericAxisData.xFollowingError		:= FALSE;
			HMI_MC_GenericAxisData.xHomed				:= FALSE;
			HMI_MC_GenericAxisData.xInError				:= FALSE;
			HMI_MC_GenericAxisData.xInPosition			:= FALSE;
			HMI_MC_GenericAxisData.xPowered				:= FALSE;
			HMI_MC_GenericAxisData.xReal				:= FALSE;
			HMI_MC_GenericAxisData.xRunning				:= FALSE;
			HMI_MC_GenericAxisData.xSynchro				:= FALSE;
			HMI_MC_GenericAxisData.xTorqueError			:= FALSE;
			HMI_MC_GenericAxisData.xHmiWait				:= TRUE;
		END_IF

		xAxisInVelocityControl	:= VAR_Machine.stFillerModule.iq_astSubModuleAxis[VAR_Machine.stFillerModule.iq_stParameters.i_uiAxisSelected].iq_stStatus.q_stMainAxisStatus.q_xVelocityControl;

	ELSIF VAR_Machine.iq_stParameter.i_uiAxisSelected >= CST_OutletSubModuleHmiStart AND VAR_Machine.iq_stParameter.i_uiAxisSelected <= CST_OutletSubModuleHmiStart + CST_LastOutletModuleAxis THEN

		VAR_Machine.stOutletModule.iq_stParameters.i_uiAxisSelected	:= VAR_Machine.iq_stParameter.i_uiAxisSelected - CST_OutletSubModuleHmiStart;

		HMI_MC_GenericAxisData.uiDiagCode				:= VAR_Machine.stOutletModule.iq_astSubModuleAxis[VAR_Machine.stOutletModule.iq_stParameters.i_uiAxisSelected].iq_stStatus.q_stMainAxisStatus.q_stInfo.Diag.StatusID.Code;
		HMI_MC_GenericAxisData.iNextAx_Number;
		HMI_MC_GenericAxisData.iPrevAx_Number;
		HMI_MC_GenericAxisData.rEncoderTemperature		:= VAR_Machine.stOutletModule.iq_astSubModuleAxis[VAR_Machine.stOutletModule.iq_stParameters.i_uiAxisSelected].iq_stStatus.q_stMainAxisStatus.q_rEncoderTemperature;
		HMI_MC_GenericAxisData.rMaxTorque;
		HMI_MC_GenericAxisData.rLagError				:= FC_DegreeToMm(CFG_MC.Mechanical.MachineStep, VAR_Machine.stOutletModule.iq_astSubModuleAxis[VAR_Machine.stOutletModule.iq_stParameters.i_uiAxisSelected].iq_stStatus.q_stMainAxisStatus.q_rLagError, FALSE);

		HMI_MC_GenericAxisData.xMotorWithBrake			:= VAR_Machine.stOutletModule.iq_astSubModuleAxis[VAR_Machine.stOutletModule.iq_stParameters.i_uiAxisSelected].iq_stStatus.q_stMainAxisStatus.q_xMotorWithBrake;
		HMI_MC_GenericAxisData.xThirdPartMotor			:= VAR_Machine.stOutletModule.iq_astSubModuleAxis[VAR_Machine.stOutletModule.iq_stParameters.i_uiAxisSelected].iq_stStatus.q_stMainAxisStatus.q_xThirdPartyMotor;
		HMI_MC_GenericAxisData.xVelocityControl			:= VAR_Machine.stOutletModule.iq_astSubModuleAxis[VAR_Machine.stOutletModule.iq_stParameters.i_uiAxisSelected].iq_stStatus.q_stMainAxisStatus.q_xVelocityControl;
		HMI_MC_GenericAxisData.xInduction				:= VAR_Machine.stOutletModule.iq_astSubModuleAxis[VAR_Machine.stOutletModule.iq_stParameters.i_uiAxisSelected].iq_stStatus.q_stMainAxisStatus.q_xInduction;
		HMI_MC_GenericAxisData.rHomingOffset			:= VAR_Machine.stOutletModule.iq_astSubModuleAxis[VAR_Machine.stOutletModule.iq_stParameters.i_uiAxisSelected].iq_stStatus.q_stMainAxisStatus.q_rHomingOffset;

		HMI_MC_GenericAxisData.rMotorTemperature		:= VAR_Machine.stOutletModule.iq_astSubModuleAxis[VAR_Machine.stOutletModule.iq_stParameters.i_uiAxisSelected].iq_stStatus.q_stMainAxisStatus.q_rMotorTemperature;
		HMI_MC_GenericAxisData.rNextAx_Position_mm;
		HMI_MC_GenericAxisData.rPosition				:= LREAL_TO_REAL(VAR_Machine.stOutletModule.iq_astSubModuleAxis[VAR_Machine.stOutletModule.iq_stParameters.i_uiAxisSelected].iq_stStatus.q_stMainAxisStatus.q_lrPosition);
		HMI_MC_GenericAxisData.rPosition_mm				:= FC_DegreeToMm(CFG_MC.Mechanical.MachineStep, HMI_MC_GenericAxisData.rPosition, TRUE);

		HMI_MC_GenericAxisData.rPrevAx_Position_mm;
		HMI_MC_GenericAxisData.rTorque					:= LREAL_TO_REAL(VAR_Machine.stOutletModule.iq_astSubModuleAxis[VAR_Machine.stOutletModule.iq_stParameters.i_uiAxisSelected].iq_stStatus.q_stMainAxisStatus.q_lrTorque);
		HMI_MC_GenericAxisData.rVelocity				:= VAR_Machine.stOutletModule.iq_astSubModuleAxis[VAR_Machine.stOutletModule.iq_stParameters.i_uiAxisSelected].iq_stStatus.q_stMainAxisStatus.q_rVelocity * 10.0;
		HMI_MC_GenericAxisData.rSwitchValue;

		HMI_MC_GenericAxisData.rTotalPhasingOffset		:= FC_DegreeToMm(CFG_MC.Mechanical.MachineStep,VAR_Machine.stOutletModule.iq_astSubModuleAxis[VAR_Machine.stOutletModule.iq_stParameters.i_uiAxisSelected].iq_stStatus.q_stMainAxisStatus.q_rTotalOffset,FALSE);

		HMI_MC_GenericAxisData.xInitialized				:= VAR_Machine.stOutletModule.iq_astSubModuleAxis[VAR_Machine.stOutletModule.iq_stParameters.i_uiAxisSelected].iq_stStatus.q_stMainAxisStatus.q_xInitDone;

		xPhasingRunning									:= VAR_Machine.stOutletModule.iq_astSubModuleAxis[VAR_Machine.stOutletModule.iq_stParameters.i_uiAxisSelected].iq_stStatus.q_stMainAxisStatus.q_xPhasingRunning;

		IF HMI_MC_GenericAxisData.xInitialized THEN
			HMI_MC_GenericAxisData.xActive				:= VAR_Machine.stOutletModule.iq_astSubModuleAxis[VAR_Machine.stOutletModule.iq_stParameters.i_uiAxisSelected].iq_stStatus.q_stMainAxisStatus.q_xActive;
			HMI_MC_GenericAxisData.xBrakeReleased		:= VAR_Machine.stOutletModule.iq_astSubModuleAxis[VAR_Machine.stOutletModule.iq_stParameters.i_uiAxisSelected].iq_stStatus.q_stMainAxisStatus.q_xBrakeReleased;
			HMI_MC_GenericAxisData.xEnabled;
			HMI_MC_GenericAxisData.xFollowingError		:= VAR_Machine.stOutletModule.iq_astSubModuleAxis[VAR_Machine.stOutletModule.iq_stParameters.i_uiAxisSelected].iq_stStatus.q_stMainAxisStatus.q_xLagError;
			HMI_MC_GenericAxisData.xHomed				:= VAR_Machine.stOutletModule.iq_astSubModuleAxis[VAR_Machine.stOutletModule.iq_stParameters.i_uiAxisSelected].iq_stStatus.q_stMainAxisStatus.q_xIsHomed;
			HMI_MC_GenericAxisData.xInError				:= VAR_Machine.stOutletModule.iq_astSubModuleAxis[VAR_Machine.stOutletModule.iq_stParameters.i_uiAxisSelected].iq_stStatus.q_stMainAxisStatus.q_xError;
			HMI_MC_GenericAxisData.xInPosition			:= VAR_Machine.stOutletModule.iq_astSubModuleAxis[VAR_Machine.stOutletModule.iq_stParameters.i_uiAxisSelected].iq_stStatus.q_stMainAxisStatus.q_xInPosition;
			HMI_MC_GenericAxisData.xPowered				:= VAR_Machine.stOutletModule.iq_astSubModuleAxis[VAR_Machine.stOutletModule.iq_stParameters.i_uiAxisSelected].iq_stStatus.q_stMainAxisStatus.q_xPoweredOn;
			HMI_MC_GenericAxisData.xReal				:= VAR_Machine.stOutletModule.iq_astSubModuleAxis[VAR_Machine.stOutletModule.iq_stParameters.i_uiAxisSelected].iq_stStatus.q_stMainAxisStatus.q_xAxisReal;
			HMI_MC_GenericAxisData.xRunning				:= NOT VAR_Machine.stOutletModule.iq_astSubModuleAxis[VAR_Machine.stOutletModule.iq_stParameters.i_uiAxisSelected].iq_stStatus.q_stMainAxisStatus.q_xStopped;
			HMI_MC_GenericAxisData.xSynchro				:= VAR_Machine.stOutletModule.iq_astSubModuleAxis[VAR_Machine.stOutletModule.iq_stParameters.i_uiAxisSelected].iq_stStatus.q_stMainAxisStatus.q_xSynchronized;
			HMI_MC_GenericAxisData.xTorqueError			:= VAR_Machine.stOutletModule.iq_astSubModuleAxis[VAR_Machine.stOutletModule.iq_stParameters.i_uiAxisSelected].iq_stStatus.q_stMainAxisStatus.q_xTorqueError;
			HMI_MC_GenericAxisData.xHmiWait				:= FALSE;
		ELSE
			HMI_MC_GenericAxisData.xActive				:= FALSE;
			HMI_MC_GenericAxisData.xBrakeReleased		:= FALSE;
			HMI_MC_GenericAxisData.xEnabled;
			HMI_MC_GenericAxisData.xFollowingError		:= FALSE;
			HMI_MC_GenericAxisData.xHomed				:= FALSE;
			HMI_MC_GenericAxisData.xInError				:= FALSE;
			HMI_MC_GenericAxisData.xInPosition			:= FALSE;
			HMI_MC_GenericAxisData.xPowered				:= FALSE;
			HMI_MC_GenericAxisData.xReal				:= FALSE;
			HMI_MC_GenericAxisData.xRunning				:= FALSE;
			HMI_MC_GenericAxisData.xSynchro				:= FALSE;
			HMI_MC_GenericAxisData.xTorqueError			:= FALSE;
			HMI_MC_GenericAxisData.xHmiWait				:= TRUE;
		END_IF

		xAxisInVelocityControl	:= VAR_Machine.stOutletModule.iq_astSubModuleAxis[VAR_Machine.stOutletModule.iq_stParameters.i_uiAxisSelected].iq_stStatus.q_stMainAxisStatus.q_xVelocityControl;

	ELSIF VAR_Machine.iq_stParameter.i_uiAxisSelected >= CST_InletSubModuleHmiStart AND VAR_Machine.iq_stParameter.i_uiAxisSelected <= CST_InletSubModuleHmiStart + CST_LastInletModuleAxis THEN

		VAR_Machine.stInletModule.iq_stParameters.i_uiAxisSelected	:= VAR_Machine.iq_stParameter.i_uiAxisSelected - CST_InletSubModuleHmiStart;

		HMI_MC_GenericAxisData.uiDiagCode				:= VAR_Machine.stInletModule.iq_astSubModuleAxis[VAR_Machine.stInletModule.iq_stParameters.i_uiAxisSelected].iq_stStatus.q_stMainAxisStatus.q_stInfo.Diag.StatusID.Code;
		HMI_MC_GenericAxisData.iNextAx_Number;
		HMI_MC_GenericAxisData.iPrevAx_Number;
		HMI_MC_GenericAxisData.rEncoderTemperature		:= VAR_Machine.stInletModule.iq_astSubModuleAxis[VAR_Machine.stInletModule.iq_stParameters.i_uiAxisSelected].iq_stStatus.q_stMainAxisStatus.q_rEncoderTemperature;
		HMI_MC_GenericAxisData.rMaxTorque;
		HMI_MC_GenericAxisData.rLagError				:= FC_DegreeToMm(CFG_MC.Mechanical.MachineStep, VAR_Machine.stInletModule.iq_astSubModuleAxis[VAR_Machine.stInletModule.iq_stParameters.i_uiAxisSelected].iq_stStatus.q_stMainAxisStatus.q_rLagError, FALSE);

		HMI_MC_GenericAxisData.xMotorWithBrake			:= VAR_Machine.stInletModule.iq_astSubModuleAxis[VAR_Machine.stInletModule.iq_stParameters.i_uiAxisSelected].iq_stStatus.q_stMainAxisStatus.q_xMotorWithBrake;
		HMI_MC_GenericAxisData.xThirdPartMotor			:= VAR_Machine.stInletModule.iq_astSubModuleAxis[VAR_Machine.stInletModule.iq_stParameters.i_uiAxisSelected].iq_stStatus.q_stMainAxisStatus.q_xThirdPartyMotor;
		HMI_MC_GenericAxisData.xVelocityControl			:= VAR_Machine.stInletModule.iq_astSubModuleAxis[VAR_Machine.stInletModule.iq_stParameters.i_uiAxisSelected].iq_stStatus.q_stMainAxisStatus.q_xVelocityControl;
		HMI_MC_GenericAxisData.xInduction				:= VAR_Machine.stInletModule.iq_astSubModuleAxis[VAR_Machine.stInletModule.iq_stParameters.i_uiAxisSelected].iq_stStatus.q_stMainAxisStatus.q_xInduction;
		HMI_MC_GenericAxisData.rHomingOffset			:= VAR_Machine.stInletModule.iq_astSubModuleAxis[VAR_Machine.stInletModule.iq_stParameters.i_uiAxisSelected].iq_stStatus.q_stMainAxisStatus.q_rHomingOffset;

		HMI_MC_GenericAxisData.rMotorTemperature		:= VAR_Machine.stInletModule.iq_astSubModuleAxis[VAR_Machine.stInletModule.iq_stParameters.i_uiAxisSelected].iq_stStatus.q_stMainAxisStatus.q_rMotorTemperature;
		HMI_MC_GenericAxisData.rNextAx_Position_mm;
		HMI_MC_GenericAxisData.rPosition				:= LREAL_TO_REAL(VAR_Machine.stInletModule.iq_astSubModuleAxis[VAR_Machine.stInletModule.iq_stParameters.i_uiAxisSelected].iq_stStatus.q_stMainAxisStatus.q_lrPosition);
		HMI_MC_GenericAxisData.rPosition_mm				:= FC_DegreeToMm(CFG_MC.Mechanical.MachineStep, HMI_MC_GenericAxisData.rPosition, TRUE);

		HMI_MC_GenericAxisData.rPrevAx_Position_mm;
		HMI_MC_GenericAxisData.rTorque					:= LREAL_TO_REAL(VAR_Machine.stInletModule.iq_astSubModuleAxis[VAR_Machine.stInletModule.iq_stParameters.i_uiAxisSelected].iq_stStatus.q_stMainAxisStatus.q_lrTorque);
		HMI_MC_GenericAxisData.rVelocity				:= VAR_Machine.stInletModule.iq_astSubModuleAxis[VAR_Machine.stInletModule.iq_stParameters.i_uiAxisSelected].iq_stStatus.q_stMainAxisStatus.q_rVelocity * 10.0;
		HMI_MC_GenericAxisData.rSwitchValue;

		HMI_MC_GenericAxisData.rTotalPhasingOffset		:= FC_DegreeToMm(CFG_MC.Mechanical.MachineStep,VAR_Machine.stInletModule.iq_astSubModuleAxis[VAR_Machine.stInletModule.iq_stParameters.i_uiAxisSelected].iq_stStatus.q_stMainAxisStatus.q_rTotalOffset,FALSE);

		HMI_MC_GenericAxisData.xInitialized				:= VAR_Machine.stInletModule.iq_astSubModuleAxis[VAR_Machine.stInletModule.iq_stParameters.i_uiAxisSelected].iq_stStatus.q_stMainAxisStatus.q_xInitDone;

		xPhasingRunning									:= VAR_Machine.stInletModule.iq_astSubModuleAxis[VAR_Machine.stInletModule.iq_stParameters.i_uiAxisSelected].iq_stStatus.q_stMainAxisStatus.q_xPhasingRunning;

		IF HMI_MC_GenericAxisData.xInitialized THEN
			HMI_MC_GenericAxisData.xActive				:= VAR_Machine.stInletModule.iq_astSubModuleAxis[VAR_Machine.stInletModule.iq_stParameters.i_uiAxisSelected].iq_stStatus.q_stMainAxisStatus.q_xActive;
			HMI_MC_GenericAxisData.xBrakeReleased		:= VAR_Machine.stInletModule.iq_astSubModuleAxis[VAR_Machine.stInletModule.iq_stParameters.i_uiAxisSelected].iq_stStatus.q_stMainAxisStatus.q_xBrakeReleased;
			HMI_MC_GenericAxisData.xEnabled;
			HMI_MC_GenericAxisData.xFollowingError		:= VAR_Machine.stInletModule.iq_astSubModuleAxis[VAR_Machine.stInletModule.iq_stParameters.i_uiAxisSelected].iq_stStatus.q_stMainAxisStatus.q_xLagError;
			HMI_MC_GenericAxisData.xHomed				:= VAR_Machine.stInletModule.iq_astSubModuleAxis[VAR_Machine.stInletModule.iq_stParameters.i_uiAxisSelected].iq_stStatus.q_stMainAxisStatus.q_xIsHomed;
			HMI_MC_GenericAxisData.xInError				:= VAR_Machine.stInletModule.iq_astSubModuleAxis[VAR_Machine.stInletModule.iq_stParameters.i_uiAxisSelected].iq_stStatus.q_stMainAxisStatus.q_xError;
			HMI_MC_GenericAxisData.xInPosition			:= VAR_Machine.stInletModule.iq_astSubModuleAxis[VAR_Machine.stInletModule.iq_stParameters.i_uiAxisSelected].iq_stStatus.q_stMainAxisStatus.q_xInPosition;
			HMI_MC_GenericAxisData.xPowered				:= VAR_Machine.stInletModule.iq_astSubModuleAxis[VAR_Machine.stInletModule.iq_stParameters.i_uiAxisSelected].iq_stStatus.q_stMainAxisStatus.q_xPoweredOn;
			HMI_MC_GenericAxisData.xReal				:= VAR_Machine.stInletModule.iq_astSubModuleAxis[VAR_Machine.stInletModule.iq_stParameters.i_uiAxisSelected].iq_stStatus.q_stMainAxisStatus.q_xAxisReal;
			HMI_MC_GenericAxisData.xRunning				:= NOT VAR_Machine.stInletModule.iq_astSubModuleAxis[VAR_Machine.stInletModule.iq_stParameters.i_uiAxisSelected].iq_stStatus.q_stMainAxisStatus.q_xStopped;
			HMI_MC_GenericAxisData.xSynchro				:= VAR_Machine.stInletModule.iq_astSubModuleAxis[VAR_Machine.stInletModule.iq_stParameters.i_uiAxisSelected].iq_stStatus.q_stMainAxisStatus.q_xSynchronized;
			HMI_MC_GenericAxisData.xTorqueError			:= VAR_Machine.stInletModule.iq_astSubModuleAxis[VAR_Machine.stInletModule.iq_stParameters.i_uiAxisSelected].iq_stStatus.q_stMainAxisStatus.q_xTorqueError;
			HMI_MC_GenericAxisData.xHmiWait				:= FALSE;
		ELSE
			HMI_MC_GenericAxisData.xActive				:= FALSE;
			HMI_MC_GenericAxisData.xBrakeReleased		:= FALSE;
			HMI_MC_GenericAxisData.xEnabled;
			HMI_MC_GenericAxisData.xFollowingError		:= FALSE;
			HMI_MC_GenericAxisData.xHomed				:= FALSE;
			HMI_MC_GenericAxisData.xInError				:= FALSE;
			HMI_MC_GenericAxisData.xInPosition			:= FALSE;
			HMI_MC_GenericAxisData.xPowered				:= FALSE;
			HMI_MC_GenericAxisData.xReal				:= FALSE;
			HMI_MC_GenericAxisData.xRunning				:= FALSE;
			HMI_MC_GenericAxisData.xSynchro				:= FALSE;
			HMI_MC_GenericAxisData.xTorqueError			:= FALSE;
			HMI_MC_GenericAxisData.xHmiWait				:= TRUE;
		END_IF

		xAxisInVelocityControl	:= VAR_Machine.stInletModule.iq_astSubModuleAxis[VAR_Machine.stInletModule.iq_stParameters.i_uiAxisSelected].iq_stStatus.q_stMainAxisStatus.q_xVelocityControl;

	ELSIF VAR_Machine.iq_stParameter.i_uiAxisSelected = CST_MachinePhasingOffset THEN

		VAR_Machine.stMasterModule.iq_stParameters.i_uiAxisSelected	:=	VAR_Machine.iq_stParameter.i_uiAxisSelected;

		HMI_MC_GenericAxisData.uiDiagCode				:= VAR_Machine.stMasterModule.iq_astSubModuleAxis[CST_MachineMasterAxis].iq_stStatus.q_stMainAxisStatus.q_stInfo.Diag.StatusID.Code;
		HMI_MC_GenericAxisData.rLagError				:= FC_DegreeToMm(CFG_MC.Mechanical.MachineStep, VAR_Machine.stMasterModule.iq_astSubModuleAxis[CST_MachineMasterAxis].iq_stStatus.q_stMainAxisStatus.q_rLagError,FALSE);

		HMI_MC_GenericAxisData.xMotorWithBrake			:= VAR_Machine.stMasterModule.iq_astSubModuleAxis[CST_MachineMasterAxis].iq_stStatus.q_stMainAxisStatus.q_xMotorWithBrake;
		HMI_MC_GenericAxisData.xThirdPartMotor			:= VAR_Machine.stMasterModule.iq_astSubModuleAxis[CST_MachineMasterAxis].iq_stStatus.q_stMainAxisStatus.q_xThirdPartyMotor;
		HMI_MC_GenericAxisData.xVelocityControl			:= VAR_Machine.stMasterModule.iq_astSubModuleAxis[CST_MachineMasterAxis].iq_stStatus.q_stMainAxisStatus.q_xVelocityControl;
		HMI_MC_GenericAxisData.xInduction				:= VAR_Machine.stMasterModule.iq_astSubModuleAxis[CST_MachineMasterAxis].iq_stStatus.q_stMainAxisStatus.q_xInduction;
		HMI_MC_GenericAxisData.rHomingOffset			:= VAR_Machine.stMasterModule.iq_astSubModuleAxis[CST_MachineMasterAxis].iq_stStatus.q_stMainAxisStatus.q_rHomingOffset;

		HMI_MC_GenericAxisData.rPosition				:= LREAL_TO_REAL(VAR_Machine.stMasterModule.iq_astSubModuleAxis[CST_MachineMasterAxis].iq_stStatus.q_stMainAxisStatus.q_lrPosition);
		HMI_MC_GenericAxisData.rPosition_mm				:= FC_DegreeToMm(CFG_MC.Mechanical.MachineStep,HMI_MC_GenericAxisData.rPosition,TRUE);

		HMI_MC_GenericAxisData.rVelocity				:= VAR_Machine.stMasterModule.iq_astSubModuleAxis[CST_MachineMasterAxis].iq_stStatus.q_stMainAxisStatus.q_rVelocity * 10.0;

		HMI_MC_GenericAxisData.rTotalPhasingOffset		:= FC_DegreeToMm(CFG_MC.Mechanical.MachineStep,VAR_Machine.stMasterModule.iq_astSubModuleAxis[CST_MachineMasterAxis].iq_stStatus.q_stMainAxisStatus.q_rTotalOffset,FALSE);

		HMI_MC_GenericAxisData.xInitialized				:= VAR_Machine.stMasterModule.iq_astSubModuleAxis[CST_MachineMasterAxis].iq_stStatus.q_stMainAxisStatus.q_xInitDone;

		xPhasingRunning									:= VAR_Machine.stMasterModule.iq_astSubModuleAxis[CST_MachineMasterAxis].iq_stStatus.q_stMainAxisStatus.q_xPhasingRunning;

		IF HMI_MC_GenericAxisData.xInitialized THEN
			HMI_MC_GenericAxisData.xActive				:= VAR_Machine.stMasterModule.iq_astSubModuleAxis[CST_MachineMasterAxis].iq_stStatus.q_stMainAxisStatus.q_xActive;
			HMI_MC_GenericAxisData.xBrakeReleased		:= FALSE;
			HMI_MC_GenericAxisData.xEnabled;
			HMI_MC_GenericAxisData.xFollowingError		:= FALSE;
			HMI_MC_GenericAxisData.xHomed				:= FALSE;
			HMI_MC_GenericAxisData.xInError				:= VAR_Machine.stMasterModule.iq_astSubModuleAxis[CST_MachineMasterAxis].iq_stStatus.q_stMainAxisStatus.q_xError;
			HMI_MC_GenericAxisData.xInPosition			:= VAR_Machine.stMasterModule.iq_astSubModuleAxis[CST_MachineMasterAxis].iq_stStatus.q_stMainAxisStatus.q_xInPosition;
			HMI_MC_GenericAxisData.xPowered				:= FALSE;
			HMI_MC_GenericAxisData.xReal				:= FALSE;
			HMI_MC_GenericAxisData.xRunning				:= FALSE;
			HMI_MC_GenericAxisData.xSynchro				:= VAR_Machine.stMasterModule.iq_astSubModuleAxis[CST_MachineMasterAxis].iq_stStatus.q_stMainAxisStatus.q_xSynchronized;
			HMI_MC_GenericAxisData.xTorqueError			:= FALSE;
			HMI_MC_GenericAxisData.xHmiWait				:= FALSE;
		ELSE
			HMI_MC_GenericAxisData.xActive				:= FALSE;
			HMI_MC_GenericAxisData.xBrakeReleased		:= FALSE;
			HMI_MC_GenericAxisData.xEnabled;
			HMI_MC_GenericAxisData.xFollowingError		:= FALSE;
			HMI_MC_GenericAxisData.xHomed				:= FALSE;
			HMI_MC_GenericAxisData.xInError				:= FALSE;
			HMI_MC_GenericAxisData.xInPosition			:= FALSE;
			HMI_MC_GenericAxisData.xPowered				:= FALSE;
			HMI_MC_GenericAxisData.xReal				:= FALSE;
			HMI_MC_GenericAxisData.xRunning				:= FALSE;
			HMI_MC_GenericAxisData.xSynchro				:= FALSE;
			HMI_MC_GenericAxisData.xTorqueError			:= FALSE;
			HMI_MC_GenericAxisData.xHmiWait				:= TRUE;
		END_IF

		xAxisInVelocityControl	:=	 VAR_Machine.stMasterModule.iq_astSubModuleAxis[CST_MachineMasterAxis].iq_stStatus.q_stMainAxisStatus.q_xVelocityControl;
	END_IF

	CASE VAR_Machine.iq_stParameter.i_uiAxisSelected OF
		99:
			HMI_MC_GenericAxisData.usiHmiName	:= 99; //V4.A.A.1.6.13

		105:
			HMI_MC_GenericAxisData.usiHmiName	:= CFG_MC.Axes.Filler.In[10].HmiNameId;

		106:
			HMI_MC_GenericAxisData.usiHmiName	:= CFG_MC.Axes.Filler.In[9].HmiNameId;

		107:
			HMI_MC_GenericAxisData.usiHmiName	:= CFG_MC.Axes.Filler.In[8].HmiNameId;

		108:
			HMI_MC_GenericAxisData.usiHmiName	:= CFG_MC.Axes.Filler.In[7].HmiNameId;

		109:
			HMI_MC_GenericAxisData.usiHmiName	:= CFG_MC.Axes.Filler.In[6].HmiNameId;

		110:
			HMI_MC_GenericAxisData.usiHmiName	:= CFG_MC.Axes.Filler.In[5].HmiNameId;

		111:
			HMI_MC_GenericAxisData.usiHmiName	:= CFG_MC.Axes.Filler.In[4].HmiNameId;

		112:
			HMI_MC_GenericAxisData.usiHmiName	:= CFG_MC.Axes.Filler.In[3].HmiNameId;

		113:
			HMI_MC_GenericAxisData.usiHmiName	:= CFG_MC.Axes.Filler.In[2].HmiNameId;

		114:
			HMI_MC_GenericAxisData.usiHmiName	:= CFG_MC.Axes.Filler.In[1].HmiNameId;

		115:
			HMI_MC_GenericAxisData.usiHmiName	:= CFG_MC.Axes.Filler.Main.HmiNameId;

		116:
			HMI_MC_GenericAxisData.usiHmiName	:= CFG_MC.Axes.Filler.Out[1].HmiNameId;

		117:
			HMI_MC_GenericAxisData.usiHmiName	:= CFG_MC.Axes.Filler.Out[2].HmiNameId;

		118:
			HMI_MC_GenericAxisData.usiHmiName	:= CFG_MC.Axes.Filler.Out[3].HmiNameId;

		119:
			HMI_MC_GenericAxisData.usiHmiName	:= CFG_MC.Axes.Filler.Out[4].HmiNameId;

		120:
			HMI_MC_GenericAxisData.usiHmiName	:= CFG_MC.Axes.Filler.Out[5].HmiNameId;

		121:
			HMI_MC_GenericAxisData.usiHmiName	:= CFG_MC.Axes.Filler.Out[6].HmiNameId;

		211:
			HMI_MC_GenericAxisData.usiHmiName	:= CFG_MC.Axes.Inlet.In[4].HmiNameId;

		212:
			HMI_MC_GenericAxisData.usiHmiName	:= CFG_MC.Axes.Inlet.In[3].HmiNameId;

		213:
			HMI_MC_GenericAxisData.usiHmiName	:= CFG_MC.Axes.Inlet.In[2].HmiNameId;

		214:
			HMI_MC_GenericAxisData.usiHmiName	:= CFG_MC.Axes.Inlet.In[1].HmiNameId;

		215:
			HMI_MC_GenericAxisData.usiHmiName	:= CFG_MC.Axes.Inlet.Main.HmiNameId;

		216:
			HMI_MC_GenericAxisData.usiHmiName	:= CFG_MC.Axes.Inlet.Out[1].HmiNameId;

		217:
			HMI_MC_GenericAxisData.usiHmiName	:= CFG_MC.Axes.Inlet.Out[2].HmiNameId;

		218:
			HMI_MC_GenericAxisData.usiHmiName	:= CFG_MC.Axes.Inlet.Out[3].HmiNameId;

		219:
			HMI_MC_GenericAxisData.usiHmiName	:= CFG_MC.Axes.Inlet.Out[4].HmiNameId;

		311:
			HMI_MC_GenericAxisData.usiHmiName	:= CFG_MC.Axes.Outlet.In[4].HmiNameId;

		312:
			HMI_MC_GenericAxisData.usiHmiName	:= CFG_MC.Axes.Outlet.In[3].HmiNameId;

		313:
			HMI_MC_GenericAxisData.usiHmiName	:= CFG_MC.Axes.Outlet.In[2].HmiNameId;

		314:
			HMI_MC_GenericAxisData.usiHmiName	:= CFG_MC.Axes.Outlet.In[1].HmiNameId;

		315:
			HMI_MC_GenericAxisData.usiHmiName	:= CFG_MC.Axes.Outlet.Main.HmiNameId;

		316:
			HMI_MC_GenericAxisData.usiHmiName	:= CFG_MC.Axes.Outlet.Out[1].HmiNameId;

		317:
			HMI_MC_GenericAxisData.usiHmiName	:= CFG_MC.Axes.Outlet.Out[2].HmiNameId;

		318:
			HMI_MC_GenericAxisData.usiHmiName	:= CFG_MC.Axes.Outlet.Out[3].HmiNameId;

		319:
			HMI_MC_GenericAxisData.usiHmiName	:= CFG_MC.Axes.Outlet.Out[4].HmiNameId;
		ELSE
			HMI_MC_GenericAxisData.usiHmiName		:= 0;
	END_CASE

	HMI_MC_AxisPresent;

	//Transfer Wheel - Encoder Diagnostic
	HMI_MC_EncoderDiagnostic.Present 	:= CFG_MC.Generic.SyncroPar.ExternalEncoder;
	HMI_MC_EncoderDiagnostic.ModuleOK 	:= MC_InputOutput.Network.Machine.Commands.MasterEncoderPositionValid;
	HMI_MC_EncoderDiagnostic.Value 		:= ITC_Motion_ExtEnc;
END_ACTION
```

#### Itc_Machine.st
```iecst
ACTION MachineInput:
	(* Reset Command To All Submodules *)
	VAR_Machine.stMasterModule.iq_stCmd.i_xReset	:= MC_InputOutput.Network.Machine.Commands.AlarmReset;
	VAR_Machine.stFillerModule.iq_stCmd.i_xReset	:= MC_InputOutput.Network.Machine.Commands.AlarmReset;
	VAR_Machine.stInletModule.iq_stCmd.i_xReset		:= MC_InputOutput.Network.Machine.Commands.AlarmReset;
	VAR_Machine.stOutletModule.iq_stCmd.i_xReset	:= MC_InputOutput.Network.Machine.Commands.AlarmReset;
	VAR_Machine.iq_stCmd.i_xReset					:= MC_InputOutput.Network.Machine.Commands.AlarmReset;

	(* Mode request from ITC *)
	VAR_Machine.iq_stCmd.i_xOnePitchShift			:= MC_InputOutput.Network.Machine.Commands.OnePitchShiftCommand;
	VAR_Machine.iq_stCmd.i_xAuto					:= MC_InputOutput.Network.Machine.Commands.AutoModalityRequest;
	VAR_Machine.iq_stCmd.i_xCombi					:= MC_InputOutput.Network.Machine.Commands.AutoCombiModalityRequest;
	VAR_Machine.iq_stCmd.i_xCombiSynchroStop		:= MC_InputOutput.Network.Machine.Commands.CombiSynchroStop;
	VAR_Machine.iq_stCmd.i_xOkToDisengage			:= MC_InputOutput.Network.Machine.Commands.OkToDisengage;
	VAR_Machine.iq_stCmd.i_xAxisPhaseShift			:= MC_InputOutput.Network.Machine.Commands.InMotionTimerModReq;
	VAR_Machine.iq_stCmd.i_xJogMode					:= MC_InputOutput.Network.Machine.Commands.JogMachineModalityRequest;
	VAR_Machine.iq_stCmd.i_xMulti					:= MC_InputOutput.Network.Machine.Commands.MultiModalityRequest;
	VAR_Machine.iq_stCmd.i_xPositioning				:= MC_InputOutput.Network.Machine.Commands.PositioningModalityRequest;
	VAR_Machine.iq_stCmd.i_xSelectiveHoming			:= MC_InputOutput.Network.Machine.Commands.SelectiveHomeModalityRequest;
	VAR_Machine.iq_stCmd.i_xBrakeRelease			:= MC_InputOutput.Network.Machine.Commands.BrakeReleaseModalityRequest;
	VAR_Machine.iq_stCmd.i_xVelocity				:= MC_InputOutput.Network.Machine.Commands.VelocityModalityRequest;
	VAR_Machine.iq_stCmd.i_xStepByStep				:= MC_InputOutput.Network.Machine.Commands.StepByStepModalityRequest;
	VAR_Machine.iq_stCmd.i_xStepByStepSingleAxis	:= MC_InputOutput.Network.Machine.Commands.StepByStepSingleAxisModReq;//V4.A.A.1.7.0 Footbar
	VAR_Machine.iq_stCmd.i_xStepByStepSingleAxisReverse	:= MC_InputOutput.Network.Machine.Commands.StepByStepSingleAxisRevModReq;//v999
	VAR_Machine.iq_stCmd.i_xQuickStop				:= MC_InputOutput.Network.Machine.Commands.MachineQuickStop;

	(* Input from ITC *)
	VAR_Machine.iq_stCmd.i_xStart							:= MC_InputOutput.Network.Machine.Commands.MachineStart;
	VAR_Machine.iq_stCmd.i_xJogPushButton					:= MC_InputOutput.Network.Machine.Commands.JogPushButton;
	VAR_Machine.iq_stParameter.i_iAxisPhaseShiftDistance	:= REAL_TO_INT(MC_InputOutput.Network.Machine.Parameters.InMotionTimerValue * 10.0);
	VAR_Machine.iq_stParameter.i_uiAxisSelected				:= MC_InputOutput.Network.Machine.Parameters.AxisSelectedOnHmi;
	VAR_Machine.iq_stParameter.i_uiPositioningOffset		:= REAL_TO_UINT(MC_InputOutput.Network.Machine.Parameters.OffsetPositioning * 10.0);
	VAR_Machine.iq_stParameter.i_uiNumberOfSteps			:= MC_InputOutput.Network.Machine.Parameters.StepNumber;
	VAR_Machine.iq_stParameter.i_uiManualVelocity			:= MC_InputOutput.Network.Machine.Parameters.ManualVelocity;

	VAR_Machine.stInletModule.iq_stCmd.i_xExternalQuickStop		:= MC_InputOutput.Network.Inlet.Commands.QuickStopInletModule	OR NOT VAR_Machine.iq_stCmd.i_xMulti;
	VAR_Machine.stFillerModule.iq_stCmd.i_xExternalQuickStop	:= MC_InputOutput.Network.Filler.Commands.QuickStopFillerModule	OR NOT VAR_Machine.iq_stCmd.i_xMulti;
	VAR_Machine.stOutletModule.iq_stCmd.i_xExternalQuickStop	:= MC_InputOutput.Network.Outlet.Commands.QuickStopOutletModule	OR NOT VAR_Machine.iq_stCmd.i_xMulti;

	VAR_Machine.stMasterModule.iq_stParameters.i_rEndlessVelocity	:= MC_InputOutput.Network.Machine.Parameters.AutoSpeed / 10.0;
	VAR_Machine.stFillerModule.iq_stParameters.i_rEndlessVelocity	:= MC_InputOutput.Network.Filler.Parameters.AutoSpeedFillerModule / 10.0;
	VAR_Machine.stInletModule.iq_stParameters.i_rEndlessVelocity	:= MC_InputOutput.Network.Inlet.Parameters.AutoSpeedInletModule / 10.0;
	VAR_Machine.stOutletModule.iq_stParameters.i_rEndlessVelocity	:= MC_InputOutput.Network.Outlet.Parameters.AutoSpeedOutletModule / 10.0;

	IF VAR_Machine.iq_stStatus.q_xHomed THEN
		VAR_Machine.stMasterModule.iq_stParameters.i_rEndlessVelocity	:= LIMIT(0, VAR_Machine.stMasterModule.iq_stParameters.i_rEndlessVelocity, CFG_MC.Movements.MachineMaxSpeed / 10);
		VAR_Machine.stFillerModule.iq_stParameters.i_rEndlessVelocity	:= LIMIT(0, VAR_Machine.stFillerModule.iq_stParameters.i_rEndlessVelocity, CFG_MC.Movements.MachineMaxSpeed / 10);
		VAR_Machine.stInletModule.iq_stParameters.i_rEndlessVelocity	:= LIMIT(0, VAR_Machine.stInletModule.iq_stParameters.i_rEndlessVelocity, CFG_MC.Movements.MachineMaxSpeed / 10);
		VAR_Machine.stOutletModule.iq_stParameters.i_rEndlessVelocity	:= LIMIT(0, VAR_Machine.stOutletModule.iq_stParameters.i_rEndlessVelocity, CFG_MC.Movements.MachineMaxSpeed / 10);
	ELSE
		VAR_Machine.stMasterModule.iq_stParameters.i_rEndlessVelocity	:= LIMIT(0, VAR_Machine.stMasterModule.iq_stParameters.i_rEndlessVelocity, 0.3 *  CFG_MC.Movements.MachineMaxSpeed / 10);
		VAR_Machine.stFillerModule.iq_stParameters.i_rEndlessVelocity	:= LIMIT(0, VAR_Machine.stFillerModule.iq_stParameters.i_rEndlessVelocity, 0.3 *  CFG_MC.Movements.MachineMaxSpeed / 10);
		VAR_Machine.stInletModule.iq_stParameters.i_rEndlessVelocity	:= LIMIT(0, VAR_Machine.stInletModule.iq_stParameters.i_rEndlessVelocity, 0.3 *  CFG_MC.Movements.MachineMaxSpeed / 10);
		VAR_Machine.stOutletModule.iq_stParameters.i_rEndlessVelocity	:= LIMIT(0, VAR_Machine.stOutletModule.iq_stParameters.i_rEndlessVelocity, 0.3 *  CFG_MC.Movements.MachineMaxSpeed / 10);
	END_IF

	VAR_Machine.stMasterModule.iq_stParameters.i_rJogVelocity	:= MC_InputOutput.Network.Machine.Parameters.JogSpeed / 10.0;
	VAR_Machine.stInletModule.iq_stParameters.i_rJogVelocity	:= MC_InputOutput.Network.Machine.Parameters.JogSpeed / 10.0;
	VAR_Machine.stFillerModule.iq_stParameters.i_rJogVelocity	:= MC_InputOutput.Network.Machine.Parameters.JogSpeed / 10.0;
	VAR_Machine.stOutletModule.iq_stParameters.i_rJogVelocity	:= MC_InputOutput.Network.Machine.Parameters.JogSpeed / 10.0;

	VAR_Machine.iq_stParameter.i_uiPositioningOffset			:= REAL_TO_UINT(MC_InputOutput.Network.Machine.Parameters.OffsetPositioning * 10.0);

	VAR_Machine.stMasterModule.iq_stParameters.i_rStopPosition	:= LREAL_TO_REAL(FC_TeensOfmmToDegrees(REAL_TO_INT(MC_InputOutput.Network.Machine.Parameters.StopPosition * 10.0), CFG_MC.Mechanical.MachineStep, FALSE,	FALSE));
	VAR_Machine.stInletModule.iq_stParameters.i_rStopPosition	:= LREAL_TO_REAL(FC_TeensOfmmToDegrees(REAL_TO_INT(MC_InputOutput.Network.Machine.Parameters.StopPosition * 10.0), CFG_MC.Mechanical.MachineStep, FALSE,	FALSE));
	VAR_Machine.stFillerModule.iq_stParameters.i_rStopPosition	:= LREAL_TO_REAL(FC_TeensOfmmToDegrees(REAL_TO_INT(MC_InputOutput.Network.Machine.Parameters.StopPosition * 10.0), CFG_MC.Mechanical.MachineStep, FALSE,	FALSE));
	VAR_Machine.stOutletModule.iq_stParameters.i_rStopPosition	:= LREAL_TO_REAL(FC_TeensOfmmToDegrees(REAL_TO_INT(MC_InputOutput.Network.Machine.Parameters.StopPosition * 10.0), CFG_MC.Mechanical.MachineStep, FALSE,	FALSE));
END_ACTION

ACTION MachineOutput:
	(* Machine status *)
	MC_InputOutput.Network.Machine.Status.HandshakeOut 			:= NOT MC_InputOutput.Network.Machine.Commands.HandShakeIn;

	MC_InputOutput.Network.Machine.Status.AxisSelectedForEndless;
	MC_InputOutput.Network.Machine.Status.SpeedForAxisSelectedEndless;
	MC_InputOutput.Network.Machine.Status.EnableEndless;

	MC_InputOutput.Network.Machine.Status.MachinePitch					:= LREAL_TO_REAL(CFG_MC.Mechanical.MachineStep);
	MC_InputOutput.Network.Machine.Status.AxisNoOp						:= VAR_Machine.iq_stStatus.q_xAxisNoOp;

	MC_InputOutput.Network.Machine.Status.AutoCmdFeedback				:= VAR_Machine.iq_stStatus.q_xAutoActive 	AND VAR_Machine.stMasterModule.iq_stCmd.i_xStart;
	MC_InputOutput.Network.Machine.Status.JogCmdFeedback				:= VAR_Machine.iq_stStatus.q_xJogActive 	AND VAR_Machine.stMasterModule.iq_stCmd.i_xStart;

	MC_InputOutput.Network.Machine.Status.NoModalityActive				:= VAR_Machine.iq_stStatus.q_xNoModalityactive;
	MC_InputOutput.Network.Machine.Status.AutoCombiModalityActive		:= VAR_Machine.iq_stStatus.q_xCombiActive;
	MC_InputOutput.Network.Machine.Status.AutoModalityActive			:= VAR_Machine.iq_stStatus.q_xAutoActive;
	MC_InputOutput.Network.Machine.Status.BrakeReleaseModalityActive	:= VAR_Machine.iq_stStatus.q_xBrakeReleaseActive;
	MC_InputOutput.Network.Machine.Status.JogModalityActive				:= VAR_Machine.iq_stStatus.q_xJogActive;
	MC_InputOutput.Network.Machine.Status.MultiModalityActive			:= VAR_Machine.iq_stStatus.q_xMultiModalityActive;
	MC_InputOutput.Network.Machine.Status.PositioningModalityActive		:= VAR_Machine.iq_stStatus.q_xPositioningActive;
	MC_InputOutput.Network.Machine.Status.SelectiveHomeModalityActive	:= VAR_Machine.iq_stStatus.q_xSelHomingActive;
	MC_InputOutput.Network.Machine.Status.StepByStepModalityActive		:= VAR_Machine.iq_stStatus.q_xStepByStepActive;
	MC_InputOutput.Network.Machine.Status.StepByStepSingleAxisModeActive:= VAR_Machine.iq_stStatus.q_xStepByStepSingleAxisActive;//V4.A.A.1.7.0
	MC_InputOutput.Network.Machine.Status.StepByStepSingleAxisRevModActive	:= VAR_Machine.iq_stStatus.q_xStepByStepSingAxisRevActive;//V999
	MC_InputOutput.Network.Machine.Status.VelocityModalityActive		:= VAR_Machine.iq_stStatus.q_xVelocityActive;
	MC_InputOutput.Network.Machine.Status.EndlessModalityActive;
	MC_InputOutput.Network.Machine.Status.ThirdPartMotStatSetupModAct;
	MC_InputOutput.Network.Machine.Status.ThirdPartMotDynSetupModAct	:= VAR_Machine.iq_stStatus.q_xThirdPartyDynSetupActive;
	MC_InputOutput.Network.Machine.Status.InductionMotSetupActive		:= VAR_Machine.iq_stStatus.q_xInductionSetupActive;

	MC_InputOutput.Network.Machine.Status.CombiFixedSpeed				:= VAR_Machine.iq_stStatus.q_xCombiFixedSpeed;
	MC_InputOutput.Network.Machine.Status.CombiSynchroInProgress		:= VAR_Machine.iq_stStatus.q_xCombiSynchroInProgress;
	MC_InputOutput.Network.Machine.Status.CombiSynchronized				:= VAR_Machine.iq_stStatus.q_xCombiSynchronized;
	MC_InputOutput.Network.Machine.Status.CombiSynchroStopDone			:= VAR_Machine.iq_stStatus.q_xCombiSynchroStopDone;
	MC_InputOutput.Network.Machine.Status.MachineHomed					:= VAR_Machine.iq_stStatus.q_xHomed;
	MC_InputOutput.Network.Machine.Status.MachineIE						:= VAR_Machine.stFillerModule.iq_stStatus.q_xModulePowered
																			AND (VAR_Machine.stOutletModule.iq_stStatus.q_xModulePowered	OR NOT VAR_Machine.stOutletModule.iq_stStatus.q_xModulePowered)
																			AND (VAR_Machine.stInletModule.iq_stStatus.q_xModulePowered		OR NOT VAR_Machine.stInletModule.iq_stStatus.q_xModulePowered);
	MC_InputOutput.Network.Machine.Status.MachineInPosition				:= VAR_Machine.iq_stStatus.q_xInPosition;
	MC_InputOutput.Network.Machine.Status.MachinePowered				:= VAR_Machine.iq_stStatus.q_xPowered;
	MC_InputOutput.Network.Machine.Status.MachineRunning				:=	NOT VAR_Machine.iq_stStatus.q_xMachineStopped;
	MC_InputOutput.Network.Machine.Status.MachineSynchro				:= VAR_Machine.stFillerModule.iq_stStatus.q_xModuleSynchronized
																			AND (VAR_Machine.stOutletModule.iq_stStatus.q_xModuleSynchronized 	OR NOT VAR_Machine.stOutletModule.iq_stStatus.q_xModuleReal)
																			AND (VAR_Machine.stInletModule.iq_stStatus.q_xModuleSynchronized 	OR NOT VAR_Machine.stInletModule.iq_stStatus.q_xModuleReal);

	MC_InputOutput.Network.Machine.Status.InMotionTimerDone		:= VAR_Machine.iq_stStatus.q_xInMotionTimerDone;

	tofShiftDoneOff(IN := MC_InputOutput.Network.Machine.Status.InMotionTimerDone OR VAR_Machine.iq_stCmd.i_xAxisPhaseShift, PT := t#10s);

	MC_InputOutput.Network.Machine.Status.ModuleNotInitialized			:= NOT VAR_Machine.stMasterModule.iq_stStatus.q_xInitDone AND NOT VAR_CamInitialized;//1.7.2a

	(* Button Enable *)
	MC_InputOutput.Network.Machine.Status.EnableAxisEnable				:= NOT VAR_Machine.stFillerModule.iq_stStatus.q_xModulePowered	AND
																			NOT VAR_Machine.stInletModule.iq_stStatus.q_xModulePowered	AND
																			NOT VAR_Machine.stOutletModule.iq_stStatus.q_xModulePowered;
	MC_InputOutput.Network.Machine.Status.EnableBrakeRelease 			:= VAR_Machine.stMasterModule.iq_stStatus.q_xModuleStopped		AND
																			VAR_Machine.stFillerModule.iq_stStatus.q_xModuleStopped		AND
																			NOT VAR_Machine.stFillerModule.iq_stStatus.q_xModulePowered	AND
																			(VAR_Machine.stOutletModule.iq_stStatus.q_xModuleStopped	AND
																			NOT VAR_Machine.stOutletModule.iq_stStatus.q_xModulePowered	OR NOT
																			VAR_Machine.stOutletModule.iq_stStatus.q_xModuleReal	)	AND
																			(VAR_Machine.stInletModule.iq_stStatus.q_xModuleStopped		AND
																			NOT VAR_Machine.stInletModule.iq_stStatus.q_xModulePowered	OR NOT
																			VAR_Machine.stInletModule.iq_stStatus.q_xModuleReal	);
	MC_InputOutput.Network.Machine.Status.EnableAuto					:= NOT VAR_Machine.iq_stStatus.q_xReactionActive;
	MC_InputOutput.Network.Machine.Status.EnableCombi					:= MC_InputOutput.Network.Machine.Commands.MasterEncoderPositionValid	AND
																			NOT VAR_Machine.iq_stStatus.q_xReactionActive						AND
																			VAR_Machine.iq_stStatus.q_xHomed;
	MC_InputOutput.Network.Machine.Status.EnableHoming					:= VAR_Machine.iq_stStatus.q_xMachineStopped		AND VAR_Machine.iq_stStatus.q_xNoModalityactive AND
																			NOT VAR_Machine.iq_stStatus.q_xReactionActive;

	MC_InputOutput.Network.Machine.Status.EnableInMotionTimer			:= (VAR_Machine.iq_stStatus.q_xAutoActive           OR
																			VAR_Machine.iq_stStatus.q_xCombiActive)			AND
																			NOT xPhasingRunning								AND
																			NOT VAR_Machine.iq_stStatus.q_xMachineStopped	AND
																			NOT VAR_Machine.iq_stStatus.q_xReactionActive	AND
																			NOT xAxisInVelocityControl						AND
																			NOT tofShiftDoneOff.Q;
	MC_InputOutput.Network.Machine.Status.EnableJog						:= VAR_Machine.iq_stStatus.q_xMachineStopped 		AND
																			NOT VAR_Machine.iq_stStatus.q_xReactionActive;
	MC_InputOutput.Network.Machine.Status.EnableMulti					:= VAR_Machine.iq_stStatus.q_xMachineStopped;
	MC_InputOutput.Network.Machine.Status.EnablePositioning				:= VAR_Machine.iq_stStatus.q_xMachineStopped		AND VAR_Machine.iq_stStatus.q_xNoModalityactive AND
																			NOT VAR_Machine.iq_stStatus.q_xReactionActive;
	MC_InputOutput.Network.Machine.Status.EnableSlowMotion				:= VAR_Machine.iq_stStatus.q_xMachineStopped		AND
																			VAR_Machine.iq_stStatus.q_xHomed;
	MC_InputOutput.Network.Machine.Status.EnableStart					:= (VAR_Machine.iq_stStatus.q_xAutoActive 			OR VAR_Machine.iq_stStatus.q_xMultiModalityActive 	OR VAR_Machine.iq_stStatus.q_xCombiActive) AND
																			NOT VAR_Machine.iq_stStatus.q_xReactionActive;
	MC_InputOutput.Network.Machine.Status.EnableStepByStep				:= VAR_Machine.iq_stStatus.q_xMachineStopped;
	MC_InputOutput.Network.Machine.Status.EnableVelocity				:= VAR_Machine.iq_stStatus.q_xMachineStopped		AND
																			NOT VAR_Machine.iq_stStatus.q_xReactionActive;

	MC_InputOutput.Network.Machine.Status.ThirdPartMotStatSetupButton;
	MC_InputOutput.Network.Machine.Status.ThirdPartMotDynSetupButton	:= VAR_Machine.iq_stStatus.q_xMachineStopped		AND
																			NOT VAR_Machine.iq_stStatus.q_xReactionActive;
	MC_InputOutput.Network.Machine.Status.InductionMotSetupButton		:= VAR_Machine.iq_stStatus.q_xMachineStopped		AND
																			NOT VAR_Machine.iq_stStatus.q_xReactionActive;

	(* Actual speed management *)
	IF VAR_Machine.iq_stStatus.q_xMultiModalityActive OR VAR_Machine.iq_stStatus.q_xMachineStopped OR
		NOT VAR_Machine.stFillerModule.iq_stStatus.q_xModulePowered
		OR (NOT VAR_Machine.stOutletModule.iq_stStatus.q_xModulePowered	AND VAR_Machine.stOutletModule.iq_stStatus.q_xModuleReal)
		OR (NOT VAR_Machine.stInletModule.iq_stStatus.q_xModulePowered	AND VAR_Machine.stInletModule.iq_stStatus.q_xModuleReal) THEN
		MC_InputOutput.Network.Machine.Status.ActualSpeed	:= 0.0;
	ELSE
		MC_InputOutput.Network.Machine.Status.ActualSpeed	:= 10.0 * MAX(VAR_Machine.stFillerModule.iq_stStatus.q_rVelocity, VAR_Machine.stOutletModule.iq_stStatus.q_rVelocity, VAR_Machine.stInletModule.iq_stStatus.q_rVelocity);
	END_IF

	MC_InputOutput.Network.Machine.Status.MachineMaxSpeed	:= CFG_MC.Movements.MachineMaxSpeed;

	(* Exception *)
	MC_InputOutput.Network.Machine.Exceptions.Fault								:= VAR_Machine.stMasterModule.iq_astSubModuleAxis[CST_MachineMasterAxis].iq_stStatus.q_stMainAxisStatus.q_xError;
	MC_InputOutput.Network.Machine.Exceptions.ExcessiveVelocityException		:= FALSE;
	MC_InputOutput.Network.Machine.Exceptions.ExcessiveAccException				:= FALSE;
	MC_InputOutput.Network.Machine.Exceptions.NoAxisEnabledException			:= FALSE;

	MC_InputOutput.Network.Machine.Exceptions.HmiChecksumException				:= VAR_Machine.iq_stStatus.q_xCheckSumError;
	MC_InputOutput.Network.Machine.Exceptions.DcBusLowMachineException			:= VAR_Machine.stMasterModule.iq_astSubModuleAxis[CST_MasterPowerSupply01].iq_stStatus.q_stMainAxisStatus.q_xDcBusLowVolatage	OR
																					VAR_Machine.stMasterModule.iq_astSubModuleAxis[CST_MasterPowerSupply02].iq_stStatus.q_stMainAxisStatus.q_xDcBusLowVolatage;
	MC_InputOutput.Network.Machine.Exceptions.PhaseMonitoringException			:= VAR_Machine.stMasterModule.iq_astSubModuleAxis[CST_MasterPowerSupply01].iq_stStatus.q_stMainAxisStatus.q_xPhaseMonitorFault	OR
																					VAR_Machine.stMasterModule.iq_astSubModuleAxis[CST_MasterPowerSupply02].iq_stStatus.q_stMainAxisStatus.q_xPhaseMonitorFault;
	MC_InputOutput.Network.Machine.Exceptions.PowerSupplyLowMachineException	:= VAR_Machine.stMasterModule.iq_astSubModuleAxis[CST_MasterPowerSupply01].iq_stStatus.q_stMainAxisStatus.q_xPowerSupplyVoltageWarning	OR//V1.3
																					VAR_Machine.stMasterModule.iq_astSubModuleAxis[CST_MasterPowerSupply02].iq_stStatus.q_stMainAxisStatus.q_xPowerSupplyVoltageWarning;//V1.3
	MC_InputOutput.Network.Machine.Exceptions.HomingException					:= (NOT VAR_Machine.stFillerModule.iq_stStatus.q_xModuleHomed	AND VAR_Machine.stFillerModule.iq_stStatus.q_xInitDone)		OR
																					(NOT VAR_Machine.stOutletModule.iq_stStatus.q_xModuleHomed	AND VAR_Machine.stOutletModule.iq_stStatus.q_xModuleReal	AND VAR_Machine.stOutletModule.iq_stStatus.q_xInitDone)	OR
																					(NOT VAR_Machine.stInletModule.iq_stStatus.q_xModuleHomed	AND VAR_Machine.stInletModule.iq_stStatus.q_xModuleReal		AND VAR_Machine.stInletModule.iq_stStatus.q_xInitDone);
	MC_InputOutput.Network.Machine.Exceptions.BleederException					:= VAR_Machine.stMasterModule.iq_astSubModuleAxis[CST_MasterPowerSupply01].iq_stStatus.q_stMainAxisStatus.q_xBleederFault	OR
																					VAR_Machine.stMasterModule.iq_astSubModuleAxis[CST_MasterPowerSupply02].iq_stStatus.q_stMainAxisStatus.q_xBleederFault;
	MC_InputOutput.Network.Machine.Exceptions.InitEncoderException				:= NOT MC_InputOutput.Network.Machine.Commands.MasterEncoderPositionValid;
	MC_InputOutput.Network.Machine.Exceptions.NegativeSpeedBlowerException;
	MC_InputOutput.Network.Machine.Exceptions.CombiException;
	MC_InputOutput.Network.Machine.Exceptions.StopBlowerException;
END_ACTION
```

#### Itc_Inlet.st
```iecst
ACTION InletInput:
	(* Commands *)

	VAR_Machine.stInletModule.iq_stCmd.i_xVelocityAxisStop			:= MC_InputOutput.Network.Inlet.Commands.VelocityAxisStop;

	FOR uiAxisIndex := CST_FirstInletModuleAxis TO CST_LastInletModuleAxis DO
		VAR_Machine.stInletModule.iq_astSubModuleAxis[uiAxisIndex].iq_stStatus.q_stMainAxisStatus.iq_xNotErrEncoder	:= MC_InputOutput.Safety.Inlet.Commands.AxesDiag[uiAxisIndex].DI_NotErrENC;
		VAR_Machine.stInletModule.iq_astSubModuleAxis[uiAxisIndex].iq_stStatus.q_stMainAxisStatus.iq_xOperational	:= MC_InputOutput.Safety.Inlet.Commands.AxesDiag[uiAxisIndex].DI_Operational;
		(* Parameters *)
		IF uiAxisIndex >= 15 THEN
			VAR_Machine.stInletModule.iq_astSubModuleAxis[uiAxisIndex].iq_stParam.i_rVelocityOffsetFactor	:= MC_InputOutput.Network.Inlet.Parameters.ConveyorKs / 100.0;
		ELSE
			VAR_Machine.stInletModule.iq_astSubModuleAxis[uiAxisIndex].iq_stParam.i_rVelocityOffsetFactor	:= MC_InputOutput.Network.Inlet.Parameters.ConveyorKs / 100.0;
		END_IF
	END_FOR

	VAR_Machine.stInletModule.iq_astSubModuleAxis[CST_MainAxis].iq_stParam.i_rTorqueErrorThreshold	:= MC_InputOutput.Network.Inlet.Parameters.TorqueError.Main;
	FOR uiAxisIndex := 1 TO 4 DO
		VAR_Machine.stInletModule.iq_astSubModuleAxis[(uiAxisIndex - 1) +  CST_FirstInletModuleAxis].iq_stParam.i_rTorqueErrorThreshold	:= MC_InputOutput.Network.Inlet.Parameters.TorqueError.In[uiAxisIndex];
	END_FOR

	FOR uiAxisIndex := 1 TO 4 DO
		VAR_Machine.stInletModule.iq_astSubModuleAxis[(uiAxisIndex) + CST_MainAxis].iq_stParam.i_rTorqueErrorThreshold	:= MC_InputOutput.Network.Inlet.Parameters.TorqueError.Out[uiAxisIndex];
	END_FOR
END_ACTION

ACTION InletOutput:
	(* Inlet status *)
	MC_InputOutput.Network.Inlet.Status.Velocity							:= VAR_Machine.stInletModule.iq_stStatus.q_rVelocity * 10.0;

	MC_InputOutput.Network.Inlet.Status.ModuleHomed							:= VAR_Machine.stInletModule.iq_stStatus.q_xModuleHomed;
	MC_InputOutput.Network.Inlet.Status.ModuleInPosition;
	MC_InputOutput.Network.Inlet.Status.ModulePowered						:= VAR_Machine.stInletModule.iq_stStatus.q_xModulePowered;
	MC_InputOutput.Network.Inlet.Status.ModuleReal							:= VAR_Machine.stInletModule.iq_stStatus.q_xModuleReal;
	MC_InputOutput.Network.Inlet.Status.ModuleRunning						:= SEL(VAR_Machine.iq_stStatus.q_xMultiModalityActive, VAR_Machine.iq_stStatus.q_xMachineStartFbk, VAR_Machine.stInletModule.iq_stStatus.q_xModuleStartFbk);
	MC_InputOutput.Network.Inlet.Status.ModuleNotInitialized				:= NOT VAR_Machine.stInletModule.iq_stStatus.q_xInitDone;

	MC_InputOutput.Network.Inlet.Status.AutoActive							:= VAR_Machine.stInletModule.iq_stStatus.q_xAutoMultiActive;
	MC_InputOutput.Network.Inlet.Status.ModuleJogActive						:= VAR_Machine.stInletModule.iq_stStatus.q_xJogMultiActive;
	MC_InputOutput.Network.Inlet.Status.SlowMotionActive					:= VAR_Machine.stInletModule.iq_stStatus.q_xSlowMotionActive;

	MC_InputOutput.Network.Inlet.Status.AutoCmdFeedback						:= VAR_Machine.stInletModule.iq_stStatus.q_xAutoMultiActive AND VAR_Machine.stInletModule.iq_stCmd.i_xStart;
	MC_InputOutput.Network.Inlet.Status.JogCmdFeedback						:= VAR_Machine.stInletModule.iq_stStatus.q_xJogMultiActive AND VAR_Machine.stInletModule.iq_stCmd.i_xJogPB;

	MC_InputOutput.Network.Inlet.Status.MainAxisReal						:= VAR_Machine.stInletModule.iq_astSubModuleAxis[CST_MainAxis].iq_stStatus.q_stMainAxisStatus.q_xAxisReal;
	MC_InputOutput.Network.Inlet.Status.In01Real							:= VAR_Machine.stInletModule.iq_astSubModuleAxis[CST_Inlet01].iq_stStatus.q_stMainAxisStatus.q_xAxisReal;
	MC_InputOutput.Network.Inlet.Status.In02Real							:= VAR_Machine.stInletModule.iq_astSubModuleAxis[CST_Inlet02].iq_stStatus.q_stMainAxisStatus.q_xAxisReal;
	MC_InputOutput.Network.Inlet.Status.In03Real							:= VAR_Machine.stInletModule.iq_astSubModuleAxis[CST_Inlet03].iq_stStatus.q_stMainAxisStatus.q_xAxisReal;
	MC_InputOutput.Network.Inlet.Status.In04Real							:= VAR_Machine.stInletModule.iq_astSubModuleAxis[CST_Inlet04].iq_stStatus.q_stMainAxisStatus.q_xAxisReal;

	(* Button Enable *)
	MC_InputOutput.Network.Inlet.Status.EnableAutoModality					:= NOT VAR_Machine.stInletModule.iq_stStatus.q_xReactionActive;
	MC_InputOutput.Network.Inlet.Status.EnableJogModality					:= VAR_Machine.stInletModule.iq_stStatus.q_xModuleStopped AND
	NOT VAR_Machine.stInletModule.iq_stStatus.q_xReactionActive;

	(* Exception *)
	(* Main axis exception *)
	IF VAR_Machine.stInletModule.iq_astSubModuleAxis[CST_MainAxis].iq_stStatus.q_stMainAxisStatus.q_xAxisReal THEN
		MC_InputOutput.Network.Inlet.Exceptions.MainAxisNotInOpException		:= NOT VAR_Machine.stInletModule.iq_astSubModuleAxis[CST_MainAxis].iq_stStatus.q_stMainAxisStatus.iq_xOperational;
		MC_InputOutput.Network.Inlet.Exceptions.MainAxisSafetyException			:= NOT MC_InputOutput.Safety.Inlet.Commands.AxesDiag[CST_MainAxis].DI_NotErrFUNC;
		MC_InputOutput.Network.Inlet.Exceptions.MainAxisDriveException			:= VAR_Machine.stInletModule.iq_astSubModuleAxis[CST_MainAxis].iq_stStatus.q_stMainAxisStatus.q_xError;
		MC_InputOutput.Network.Inlet.Exceptions.MainAxisTorqueException			:= VAR_Machine.stInletModule.iq_astSubModuleAxis[CST_MainAxis].iq_stStatus.q_stMainAxisStatus.q_xTorqueError;
		MC_InputOutput.Network.Inlet.Exceptions.MainAxisTrackException			:= VAR_Machine.stInletModule.iq_astSubModuleAxis[CST_MainAxis].iq_stStatus.q_stMainAxisStatus.q_xLagError;
		MC_InputOutput.Network.Inlet.Exceptions.MainAxisHomeException			:= NOT VAR_Machine.stInletModule.iq_astSubModuleAxis[CST_MainAxis].iq_stStatus.q_stMainAxisStatus.q_xIsHomed AND
																					VAR_Machine.stInletModule.iq_astSubModuleAxis[CST_MainAxis].iq_stStatus.q_stMainAxisStatus.q_xInitDone;
	END_IF

	(* Inlet axis exception *)
	IF VAR_Machine.stInletModule.iq_astSubModuleAxis[CST_Inlet01].iq_stStatus.q_stMainAxisStatus.q_xAxisReal THEN
		IF NOT CFG_MC.Axes.Inlet.In[1].VelocityControl THEN
			MC_InputOutput.Network.Inlet.Exceptions.Inlet01NotInOpException			:= NOT VAR_Machine.stInletModule.iq_astSubModuleAxis[CST_Inlet01].iq_stStatus.q_stMainAxisStatus.iq_xOperational;
			MC_InputOutput.Network.Inlet.Exceptions.Inlet01SafetyException			:= NOT MC_InputOutput.Safety.Inlet.Commands.AxesDiag[CST_Inlet01].DI_NotErrFUNC;
		END_IF
		MC_InputOutput.Network.Inlet.Exceptions.Inlet01TorqueException				:= VAR_Machine.stInletModule.iq_astSubModuleAxis[CST_Inlet01].iq_stStatus.q_stMainAxisStatus.q_xTorqueError;
		MC_InputOutput.Network.Inlet.Exceptions.Inlet01TrackException				:= VAR_Machine.stInletModule.iq_astSubModuleAxis[CST_Inlet01].iq_stStatus.q_stMainAxisStatus.q_xLagError;
		MC_InputOutput.Network.Inlet.Exceptions.Inlet01DriveException				:= VAR_Machine.stInletModule.iq_astSubModuleAxis[CST_Inlet01].iq_stStatus.q_stMainAxisStatus.q_xError;
		MC_InputOutput.Network.Inlet.Exceptions.Inlet01HomeException				:= NOT VAR_Machine.stInletModule.iq_astSubModuleAxis[CST_Inlet01].iq_stStatus.q_stMainAxisStatus.q_xIsHomed AND
																						VAR_Machine.stInletModule.iq_astSubModuleAxis[CST_Inlet01].iq_stStatus.q_stMainAxisStatus.q_xInitDone;
	END_IF

	IF VAR_Machine.stInletModule.iq_astSubModuleAxis[CST_Inlet02].iq_stStatus.q_stMainAxisStatus.q_xAxisReal THEN
		IF NOT CFG_MC.Axes.Inlet.In[2].VelocityControl THEN
			MC_InputOutput.Network.Inlet.Exceptions.Inlet02NotInOpException			:= NOT VAR_Machine.stInletModule.iq_astSubModuleAxis[CST_Inlet02].iq_stStatus.q_stMainAxisStatus.iq_xOperational;
			MC_InputOutput.Network.Inlet.Exceptions.Inlet02SafetyException			:= NOT MC_InputOutput.Safety.Inlet.Commands.AxesDiag[CST_Inlet02].DI_NotErrFUNC;
		END_IF
		MC_InputOutput.Network.Inlet.Exceptions.Inlet02TorqueException				:= VAR_Machine.stInletModule.iq_astSubModuleAxis[CST_Inlet02].iq_stStatus.q_stMainAxisStatus.q_xTorqueError;
		MC_InputOutput.Network.Inlet.Exceptions.Inlet02TrackException				:= VAR_Machine.stInletModule.iq_astSubModuleAxis[CST_Inlet02].iq_stStatus.q_stMainAxisStatus.q_xLagError;
		MC_InputOutput.Network.Inlet.Exceptions.Inlet02DriveException				:= VAR_Machine.stInletModule.iq_astSubModuleAxis[CST_Inlet02].iq_stStatus.q_stMainAxisStatus.q_xError;
		MC_InputOutput.Network.Inlet.Exceptions.Inlet02HomeException				:= NOT VAR_Machine.stInletModule.iq_astSubModuleAxis[CST_Inlet02].iq_stStatus.q_stMainAxisStatus.q_xIsHomed AND
																						VAR_Machine.stInletModule.iq_astSubModuleAxis[CST_Inlet02].iq_stStatus.q_stMainAxisStatus.q_xInitDone;
	END_IF

	IF VAR_Machine.stInletModule.iq_astSubModuleAxis[CST_Inlet03].iq_stStatus.q_stMainAxisStatus.q_xAxisReal THEN
		IF NOT CFG_MC.Axes.Inlet.In[3].VelocityControl THEN
			MC_InputOutput.Network.Inlet.Exceptions.Inlet03NotInOpException			:= NOT VAR_Machine.stInletModule.iq_astSubModuleAxis[CST_Inlet03].iq_stStatus.q_stMainAxisStatus.iq_xOperational;
			MC_InputOutput.Network.Inlet.Exceptions.Inlet03SafetyException			:= NOT MC_InputOutput.Safety.Inlet.Commands.AxesDiag[CST_Inlet03].DI_NotErrFUNC;
		END_IF
		MC_InputOutput.Network.Inlet.Exceptions.Inlet03TorqueException				:= VAR_Machine.stInletModule.iq_astSubModuleAxis[CST_Inlet03].iq_stStatus.q_stMainAxisStatus.q_xTorqueError;
		MC_InputOutput.Network.Inlet.Exceptions.Inlet03TrackException				:= VAR_Machine.stInletModule.iq_astSubModuleAxis[CST_Inlet03].iq_stStatus.q_stMainAxisStatus.q_xLagError;
		MC_InputOutput.Network.Inlet.Exceptions.Inlet03DriveException				:= VAR_Machine.stInletModule.iq_astSubModuleAxis[CST_Inlet03].iq_stStatus.q_stMainAxisStatus.q_xError;
		MC_InputOutput.Network.Inlet.Exceptions.Inlet03HomeException				:= NOT VAR_Machine.stInletModule.iq_astSubModuleAxis[CST_Inlet03].iq_stStatus.q_stMainAxisStatus.q_xIsHomed AND
																						VAR_Machine.stInletModule.iq_astSubModuleAxis[CST_Inlet03].iq_stStatus.q_stMainAxisStatus.q_xInitDone;
	END_IF

	IF VAR_Machine.stInletModule.iq_astSubModuleAxis[CST_Inlet04].iq_stStatus.q_stMainAxisStatus.q_xAxisReal THEN
		IF NOT CFG_MC.Axes.Inlet.In[4].VelocityControl THEN
			MC_InputOutput.Network.Inlet.Exceptions.Inlet04NotInOpException			:= NOT VAR_Machine.stInletModule.iq_astSubModuleAxis[CST_Inlet04].iq_stStatus.q_stMainAxisStatus.iq_xOperational;
			MC_InputOutput.Network.Inlet.Exceptions.Inlet04SafetyException			:= NOT MC_InputOutput.Safety.Inlet.Commands.AxesDiag[CST_Inlet04].DI_NotErrFUNC;
		END_IF
		MC_InputOutput.Network.Inlet.Exceptions.Inlet04DriveException				:= VAR_Machine.stInletModule.iq_astSubModuleAxis[CST_Inlet04].iq_stStatus.q_stMainAxisStatus.q_xError;
		MC_InputOutput.Network.Inlet.Exceptions.Inlet04TorqueException				:= VAR_Machine.stInletModule.iq_astSubModuleAxis[CST_Inlet04].iq_stStatus.q_stMainAxisStatus.q_xTorqueError;
		MC_InputOutput.Network.Inlet.Exceptions.Inlet04TrackException				:= VAR_Machine.stInletModule.iq_astSubModuleAxis[CST_Inlet04].iq_stStatus.q_stMainAxisStatus.q_xLagError;
		MC_InputOutput.Network.Inlet.Exceptions.Inlet04HomeException 				:= NOT VAR_Machine.stInletModule.iq_astSubModuleAxis[CST_Inlet04].iq_stStatus.q_stMainAxisStatus.q_xIsHomed AND
																						VAR_Machine.stInletModule.iq_astSubModuleAxis[CST_Inlet04].iq_stStatus.q_stMainAxisStatus.q_xInitDone;
	END_IF
END_ACTION
```
